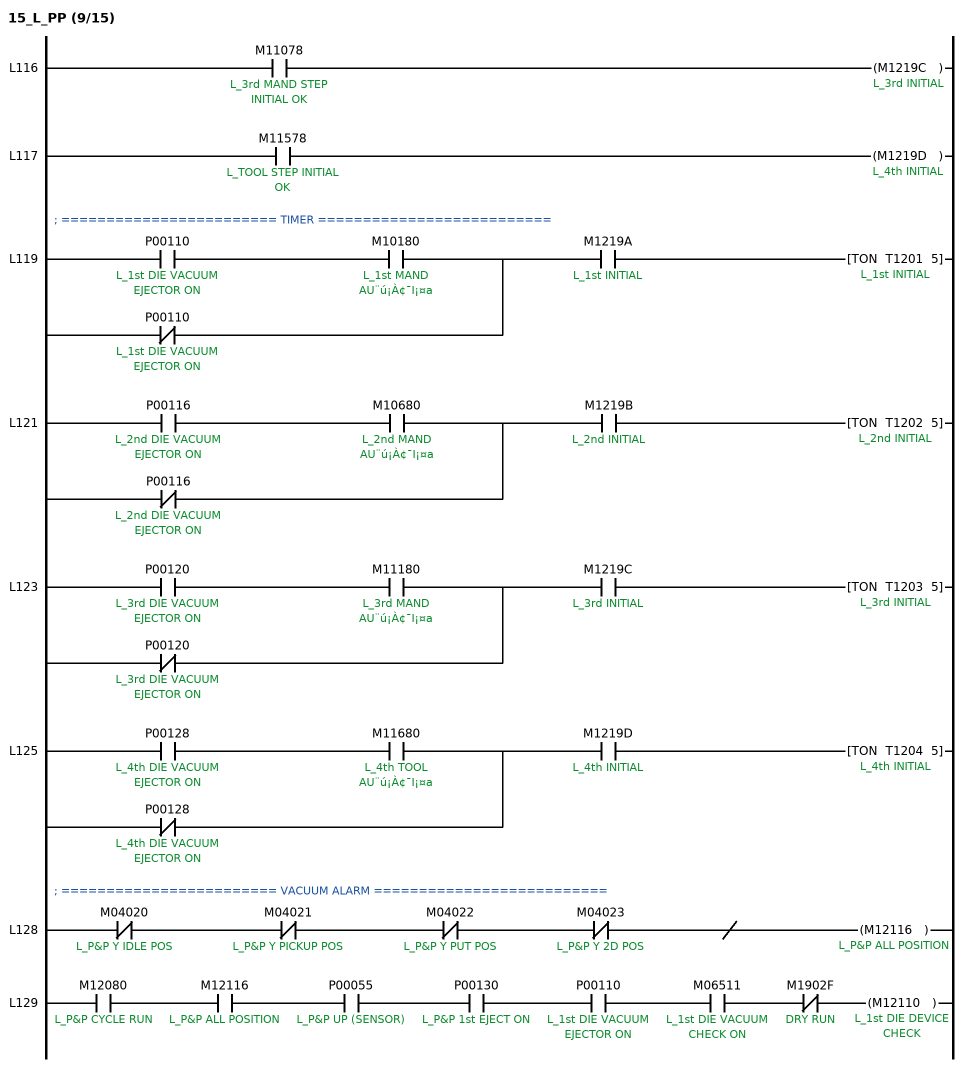
[picture p120: 15_L_PP rungs L116-L129]
; L116
LOAD      M11078	// L_3rd MAND STEP INITIAL OK
OUT       M1219C	// L_3rd INITIAL
; L117
LOAD      M11578	// L_TOOL STEP INITIAL OK
OUT       M1219D	// L_4th INITIAL
// ======================== TIMER ==========================
; L119
LOAD      P00110	// L_1st DIE VACUUM EJECTOR ON
AND       M10180	// L_1st MAND AU¨ú¡À¢¯I¡¤a
OR NOT    P00110	// L_1st DIE VACUUM EJECTOR ON
AND       M1219A	// L_1st INITIAL
TON       T1201 5	// L_1st INITIAL
; L121
LOAD      P00116	// L_2nd DIE VACUUM EJECTOR ON
AND       M10680	// L_2nd MAND AU¨ú¡À¢¯I¡¤a
OR NOT    P00116	// L_2nd DIE VACUUM EJECTOR ON
AND       M1219B	// L_2nd INITIAL
TON       T1202 5	// L_2nd INITIAL
; L123
LOAD      P00120	// L_3rd DIE VACUUM EJECTOR ON
AND       M11180	// L_3rd MAND AU¨ú¡À¢¯I¡¤a
OR NOT    P00120	// L_3rd DIE VACUUM EJECTOR ON
AND       M1219C	// L_3rd INITIAL
TON       T1203 5	// L_3rd INITIAL
; L125
LOAD      P00128	// L_4th DIE VACUUM EJECTOR ON
AND       M11680	// L_4th TOOL AU¨ú¡À¢¯I¡¤a
OR NOT    P00128	// L_4th DIE VACUUM EJECTOR ON
AND       M1219D	// L_4th INITIAL
TON       T1204 5	// L_4th INITIAL
// ======================== VACUUM ALARM ==========================
; L128
LOAD NOT  M04020	// L_P&P Y IDLE POS
AND NOT   M04021	// L_P&P Y PICKUP POS
AND NOT   M04022	// L_P&P Y PUT POS
AND NOT   M04023	// L_P&P Y 2D POS
NOT
OUT       M12116	// L_P&P ALL POSITION
; L129
LOAD      M12080	// L_P&P CYCLE RUN
AND       M12116	// L_P&P ALL POSITION
AND       P00055	// L_P&P UP (SENSOR)
AND       P00130	// L_P&P 1st EJECT ON
AND       P00110	// L_1st DIE VACUUM EJECTOR ON
AND       M06511	// L_1st DIE VACUUM CHECK ON
AND NOT   M1902F	// DRY RUN
OUT       M12110	// L_1st DIE DEVICE CHECK

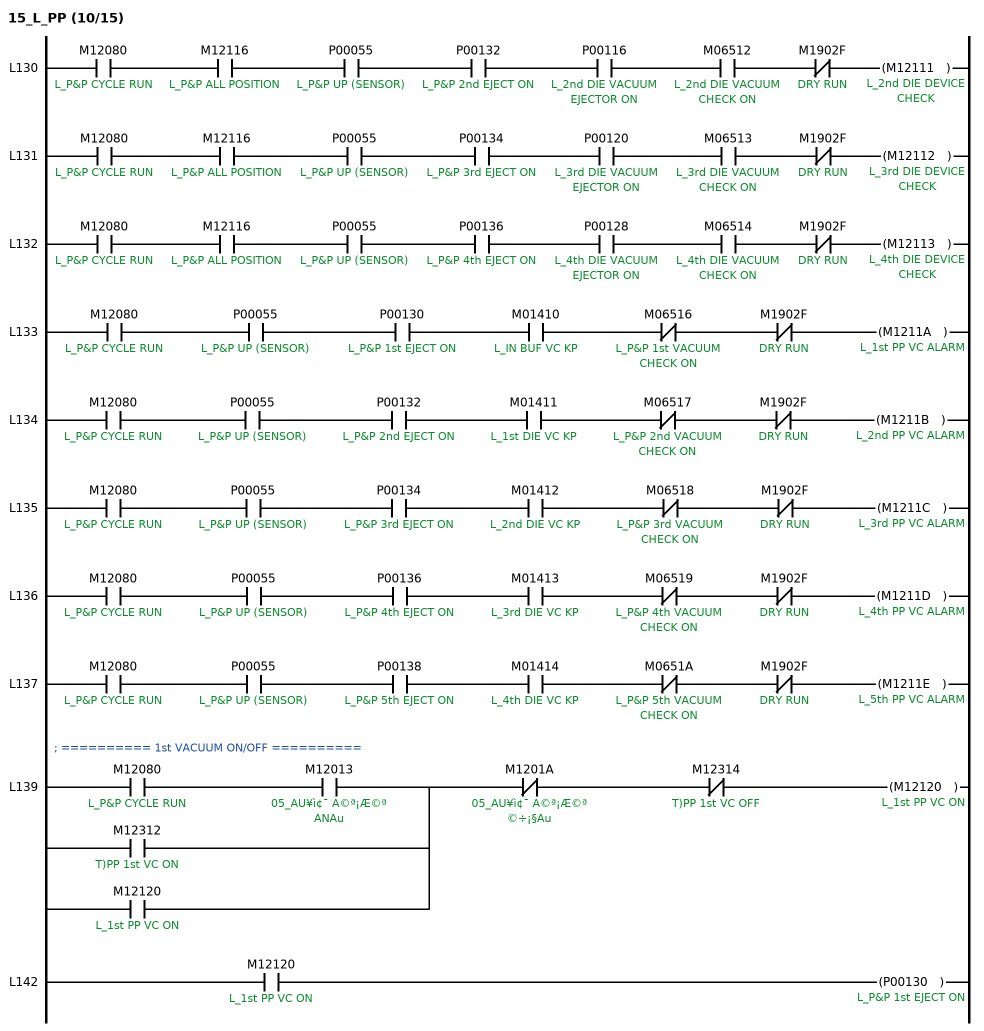
; L130
LOAD      M12080	// L_P&P CYCLE RUN
AND       M12116	// L_P&P ALL POSITION
AND       P00055	// L_P&P UP (SENSOR)
AND       P00132	// L_P&P 2nd EJECT ON
AND       P00116	// L_2nd DIE VACUUM EJECTOR ON
AND       M06512	// L_2nd DIE VACUUM CHECK ON
AND NOT   M1902F	// DRY RUN
OUT       M12111	// L_2nd DIE DEVICE CHECK
; L131
LOAD      M12080	// L_P&P CYCLE RUN
AND       M12116	// L_P&P ALL POSITION
AND       P00055	// L_P&P UP (SENSOR)
AND       P00134	// L_P&P 3rd EJECT ON
AND       P00120	// L_3rd DIE VACUUM EJECTOR ON
AND       M06513	// L_3rd DIE VACUUM CHECK ON
AND NOT   M1902F	// DRY RUN
OUT       M12112	// L_3rd DIE DEVICE CHECK
; L132
LOAD      M12080	// L_P&P CYCLE RUN
AND       M12116	// L_P&P ALL POSITION
AND       P00055	// L_P&P UP (SENSOR)
AND       P00136	// L_P&P 4th EJECT ON
AND       P00128	// L_4th DIE VACUUM EJECTOR ON
AND       M06514	// L_4th DIE VACUUM CHECK ON
AND NOT   M1902F	// DRY RUN
OUT       M12113	// L_4th DIE DEVICE CHECK
; L133
LOAD      M12080	// L_P&P CYCLE RUN
AND       P00055	// L_P&P UP (SENSOR)
AND       P00130	// L_P&P 1st EJECT ON
AND       M01410	// L_IN BUF VC KP
AND NOT   M06516	// L_P&P 1st VACUUM CHECK ON
AND NOT   M1902F	// DRY RUN
OUT       M1211A	// L_1st PP VC ALARM
; L134
LOAD      M12080	// L_P&P CYCLE RUN
AND       P00055	// L_P&P UP (SENSOR)
AND       P00132	// L_P&P 2nd EJECT ON
AND       M01411	// L_1st DIE VC KP
AND NOT   M06517	// L_P&P 2nd VACUUM CHECK ON
AND NOT   M1902F	// DRY RUN
OUT       M1211B	// L_2nd PP VC ALARM
; L135
LOAD      M12080	// L_P&P CYCLE RUN
AND       P00055	// L_P&P UP (SENSOR)
AND       P00134	// L_P&P 3rd EJECT ON
AND       M01412	// L_2nd DIE VC KP
AND NOT   M06518	// L_P&P 3rd VACUUM CHECK ON
AND NOT   M1902F	// DRY RUN
OUT       M1211C	// L_3rd PP VC ALARM
; L136
LOAD      M12080	// L_P&P CYCLE RUN
AND       P00055	// L_P&P UP (SENSOR)
AND       P00136	// L_P&P 4th EJECT ON
AND       M01413	// L_3rd DIE VC KP
AND NOT   M06519	// L_P&P 4th VACUUM CHECK ON
AND NOT   M1902F	// DRY RUN
OUT       M1211D	// L_4th PP VC ALARM
; L137
LOAD      M12080	// L_P&P CYCLE RUN
AND       P00055	// L_P&P UP (SENSOR)
AND       P00138	// L_P&P 5th EJECT ON
AND       M01414	// L_4th DIE VC KP
AND NOT   M0651A	// L_P&P 5th VACUUM CHECK ON
AND NOT   M1902F	// DRY RUN
OUT       M1211E	// L_5th PP VC ALARM
// ========== 1st VACUUM ON/OFF ==========
; L139
LOAD      M12080	// L_P&P CYCLE RUN
AND       M12013	// 05_AU¥ì¢¯ A©ª¡Æ©ª ANAu
OR        M12312	// T)PP 1st VC ON
OR        M12120	// L_1st PP VC ON
AND NOT   M1201A	// 05_AU¥ì¢¯ A©ª¡Æ©ª ©÷¡§Au
AND NOT   M12314	// T)PP 1st VC OFF
OUT       M12120	// L_1st PP VC ON
; L142
LOAD      M12120	// L_1st PP VC ON
OUT       P00130	// L_P&P 1st EJECT ON

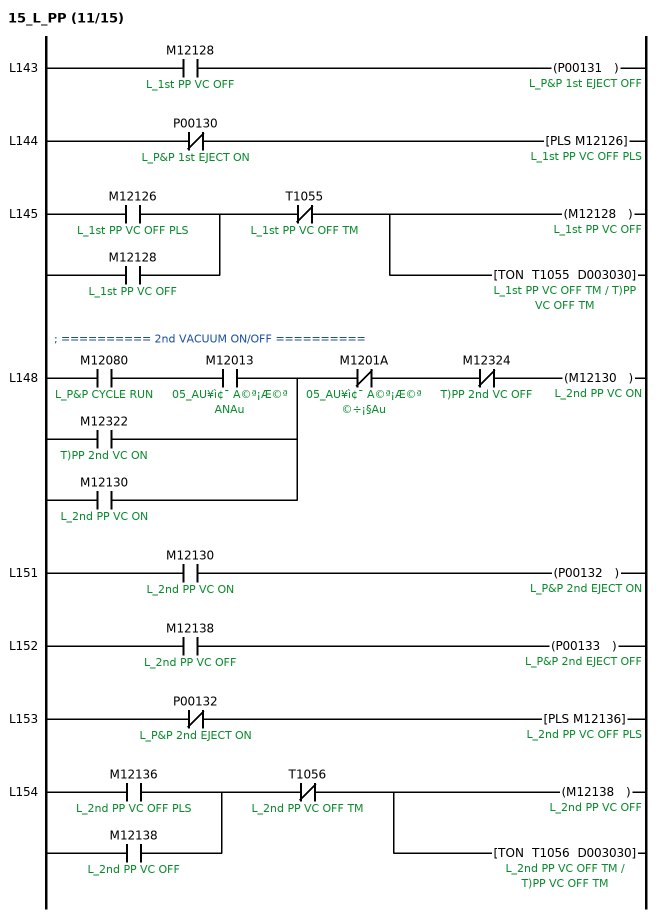
; L143
LOAD      M12128	// L_1st PP VC OFF
OUT       P00131	// L_P&P 1st EJECT OFF
; L144
LOAD NOT  P00130	// L_P&P 1st EJECT ON
OUTP      M12126	// L_1st PP VC OFF PLS
; L145
LOAD      M12126	// L_1st PP VC OFF PLS
OR        M12128	// L_1st PP VC OFF
AND NOT   T1055	// L_1st PP VC OFF TM
OUT       M12128	// L_1st PP VC OFF
TON       T1055 D003030	// L_1st PP VC OFF TM / T)PP VC OFF TM
// ========== 2nd VACUUM ON/OFF ==========
; L148
LOAD      M12080	// L_P&P CYCLE RUN
AND       M12013	// 05_AU¥ì¢¯ A©ª¡Æ©ª ANAu
OR        M12322	// T)PP 2nd VC ON
OR        M12130	// L_2nd PP VC ON
AND NOT   M1201A	// 05_AU¥ì¢¯ A©ª¡Æ©ª ©÷¡§Au
AND NOT   M12324	// T)PP 2nd VC OFF
OUT       M12130	// L_2nd PP VC ON
; L151
LOAD      M12130	// L_2nd PP VC ON
OUT       P00132	// L_P&P 2nd EJECT ON
; L152
LOAD      M12138	// L_2nd PP VC OFF
OUT       P00133	// L_P&P 2nd EJECT OFF
; L153
LOAD NOT  P00132	// L_P&P 2nd EJECT ON
OUTP      M12136	// L_2nd PP VC OFF PLS
; L154
LOAD      M12136	// L_2nd PP VC OFF PLS
OR        M12138	// L_2nd PP VC OFF
AND NOT   T1056	// L_2nd PP VC OFF TM
OUT       M12138	// L_2nd PP VC OFF
TON       T1056 D003030	// L_2nd PP VC OFF TM / T)PP VC OFF TM

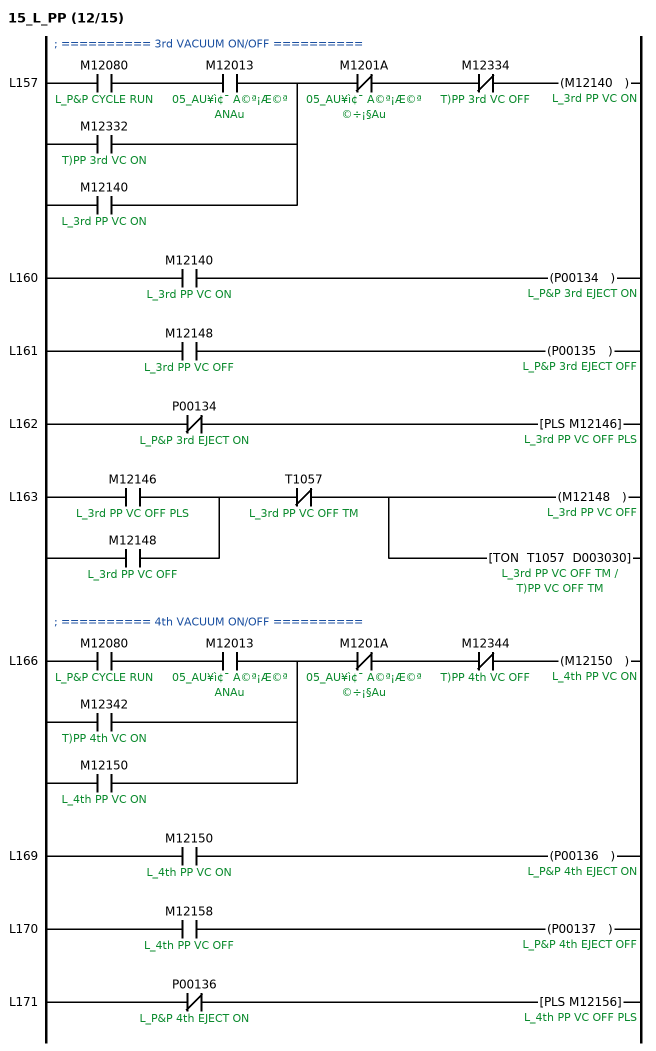
// ========== 3rd VACUUM ON/OFF ==========
; L157
LOAD      M12080	// L_P&P CYCLE RUN
AND       M12013	// 05_AU¥ì¢¯ A©ª¡Æ©ª ANAu
OR        M12332	// T)PP 3rd VC ON
OR        M12140	// L_3rd PP VC ON
AND NOT   M1201A	// 05_AU¥ì¢¯ A©ª¡Æ©ª ©÷¡§Au
AND NOT   M12334	// T)PP 3rd VC OFF
OUT       M12140	// L_3rd PP VC ON
; L160
LOAD      M12140	// L_3rd PP VC ON
OUT       P00134	// L_P&P 3rd EJECT ON
; L161
LOAD      M12148	// L_3rd PP VC OFF
OUT       P00135	// L_P&P 3rd EJECT OFF
; L162
LOAD NOT  P00134	// L_P&P 3rd EJECT ON
OUTP      M12146	// L_3rd PP VC OFF PLS
; L163
LOAD      M12146	// L_3rd PP VC OFF PLS
OR        M12148	// L_3rd PP VC OFF
AND NOT   T1057	// L_3rd PP VC OFF TM
OUT       M12148	// L_3rd PP VC OFF
TON       T1057 D003030	// L_3rd PP VC OFF TM / T)PP VC OFF TM
// ========== 4th VACUUM ON/OFF ==========
; L166
LOAD      M12080	// L_P&P CYCLE RUN
AND       M12013	// 05_AU¥ì¢¯ A©ª¡Æ©ª ANAu
OR        M12342	// T)PP 4th VC ON
OR        M12150	// L_4th PP VC ON
AND NOT   M1201A	// 05_AU¥ì¢¯ A©ª¡Æ©ª ©÷¡§Au
AND NOT   M12344	// T)PP 4th VC OFF
OUT       M12150	// L_4th PP VC ON
; L169
LOAD      M12150	// L_4th PP VC ON
OUT       P00136	// L_P&P 4th EJECT ON
; L170
LOAD      M12158	// L_4th PP VC OFF
OUT       P00137	// L_P&P 4th EJECT OFF
; L171
LOAD NOT  P00136	// L_P&P 4th EJECT ON
OUTP      M12156	// L_4th PP VC OFF PLS

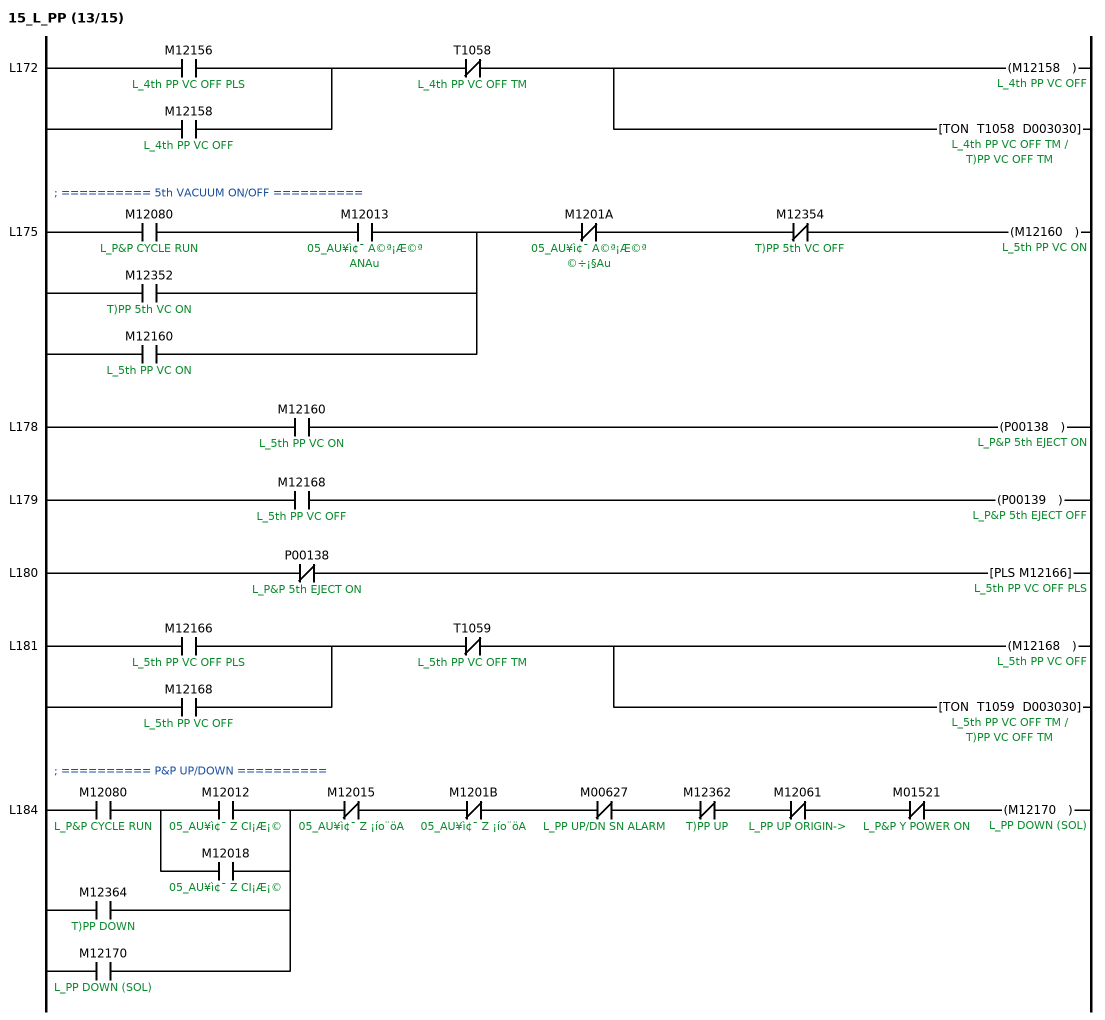
; L172
LOAD      M12156	// L_4th PP VC OFF PLS
OR        M12158	// L_4th PP VC OFF
AND NOT   T1058	// L_4th PP VC OFF TM
OUT       M12158	// L_4th PP VC OFF
TON       T1058 D003030	// L_4th PP VC OFF TM / T)PP VC OFF TM
// ========== 5th VACUUM ON/OFF ==========
; L175
LOAD      M12080	// L_P&P CYCLE RUN
AND       M12013	// 05_AU¥ì¢¯ A©ª¡Æ©ª ANAu
OR        M12352	// T)PP 5th VC ON
OR        M12160	// L_5th PP VC ON
AND NOT   M1201A	// 05_AU¥ì¢¯ A©ª¡Æ©ª ©÷¡§Au
AND NOT   M12354	// T)PP 5th VC OFF
OUT       M12160	// L_5th PP VC ON
; L178
LOAD      M12160	// L_5th PP VC ON
OUT       P00138	// L_P&P 5th EJECT ON
; L179
LOAD      M12168	// L_5th PP VC OFF
OUT       P00139	// L_P&P 5th EJECT OFF
; L180
LOAD NOT  P00138	// L_P&P 5th EJECT ON
OUTP      M12166	// L_5th PP VC OFF PLS
; L181
LOAD      M12166	// L_5th PP VC OFF PLS
OR        M12168	// L_5th PP VC OFF
AND NOT   T1059	// L_5th PP VC OFF TM
OUT       M12168	// L_5th PP VC OFF
TON       T1059 D003030	// L_5th PP VC OFF TM / T)PP VC OFF TM
// ========== P&P UP/DOWN ==========
; L184
LOAD      M12080	// L_P&P CYCLE RUN
LOAD      M12012	// 05_AU¥ì¢¯ Z CI¡Æ¡©
OR        M12018	// 05_AU¥ì¢¯ Z CI¡Æ¡©
AND LOAD
OR        M12364	// T)PP DOWN
OR        M12170	// L_PP DOWN (SOL)
AND NOT   M12015	// 05_AU¥ì¢¯ Z ¡ío¨öA
AND NOT   M1201B	// 05_AU¥ì¢¯ Z ¡ío¨öA
AND NOT   M00627	// L_PP UP/DN SN ALARM
AND NOT   M12362	// T)PP UP
AND NOT   M12061	// L_PP UP ORIGIN->
AND NOT   M01521	// L_P&P Y POWER ON
OUT       M12170	// L_PP DOWN (SOL)

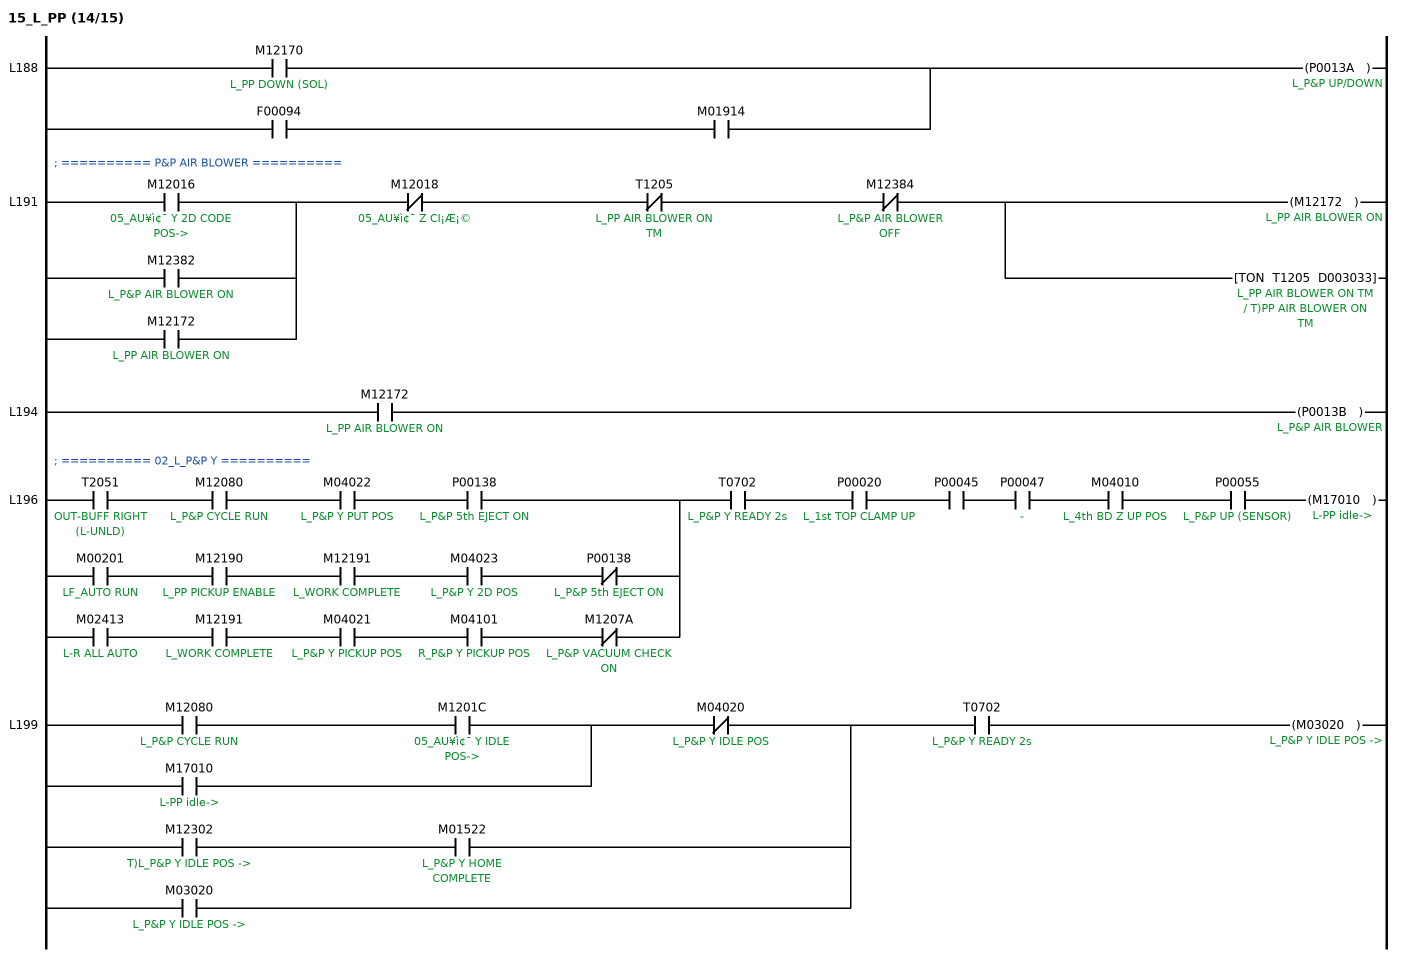
; L188
LOAD      M12170	// L_PP DOWN (SOL)
LOAD      F00094
AND       M01914
OR LOAD
OUT       P0013A	// L_P&P UP/DOWN
// ========== P&P AIR BLOWER ==========
; L191
LOAD      M12016	// 05_AU¥ì¢¯ Y 2D CODE POS->
OR        M12382	// L_P&P AIR BLOWER ON
OR        M12172	// L_PP AIR BLOWER ON
AND NOT   M12018	// 05_AU¥ì¢¯ Z CI¡Æ¡©
AND NOT   T1205	// L_PP AIR BLOWER ON TM
AND NOT   M12384	// L_P&P AIR BLOWER OFF
OUT       M12172	// L_PP AIR BLOWER ON
TON       T1205 D003033	// L_PP AIR BLOWER ON TM / T)PP AIR BLOWER ON TM
; L194
LOAD      M12172	// L_PP AIR BLOWER ON
OUT       P0013B	// L_P&P AIR BLOWER
// ========== 02_L_P&P Y ==========
; L196
LOAD      T2051	// OUT-BUFF RIGHT (L-UNLD)
AND       M12080	// L_P&P CYCLE RUN
AND       M04022	// L_P&P Y PUT POS
AND       P00138	// L_P&P 5th EJECT ON
LOAD      M00201	// LF_AUTO RUN
AND       M12190	// L_PP PICKUP ENABLE
AND       M12191	// L_WORK COMPLETE
AND       M04023	// L_P&P Y 2D POS
AND NOT   P00138	// L_P&P 5th EJECT ON
OR LOAD
LOAD      M02413	// L-R ALL AUTO
AND       M12191	// L_WORK COMPLETE
AND       M04021	// L_P&P Y PICKUP POS
AND       M04101	// R_P&P Y PICKUP POS
AND NOT   M1207A	// L_P&P VACUUM CHECK ON
OR LOAD
AND       T0702	// L_P&P Y READY 2s
AND       P00020	// L_1st TOP CLAMP UP
AND       P00045
AND       P00047	// -
AND       M04010	// L_4th BD Z UP POS
AND       P00055	// L_P&P UP (SENSOR)
OUT       M17010	// L-PP idle->
; L199
LOAD      M12080	// L_P&P CYCLE RUN
AND       M1201C	// 05_AU¥ì¢¯ Y IDLE POS->
OR        M17010	// L-PP idle->
AND NOT   M04020	// L_P&P Y IDLE POS
LOAD      M12302	// T)L_P&P Y IDLE POS ->
AND       M01522	// L_P&P Y HOME COMPLETE
OR LOAD
OR        M03020	// L_P&P Y IDLE POS ->
AND       T0702	// L_P&P Y READY 2s
OUT       M03020	// L_P&P Y IDLE POS ->

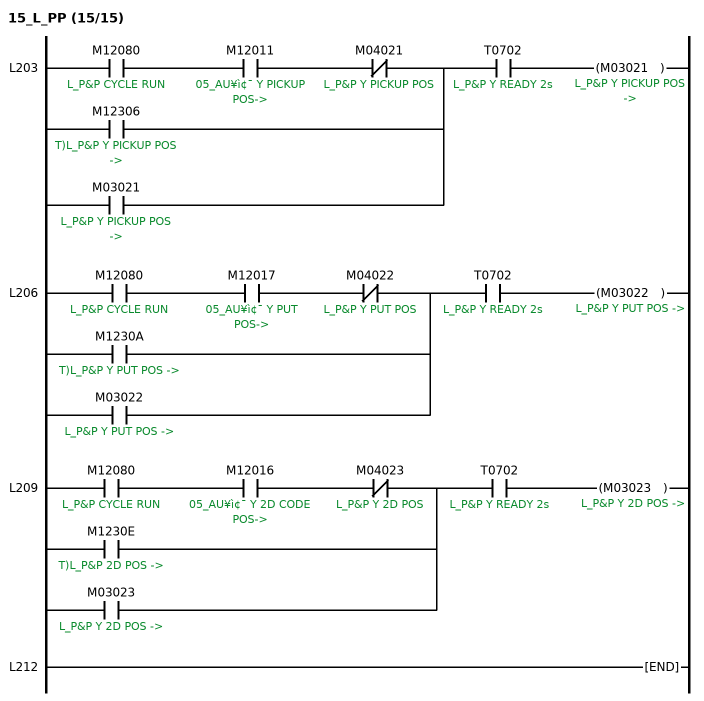
; L203
LOAD      M12080	// L_P&P CYCLE RUN
AND       M12011	// 05_AU¥ì¢¯ Y PICKUP POS->
AND NOT   M04021	// L_P&P Y PICKUP POS
OR        M12306	// T)L_P&P Y PICKUP POS ->
OR        M03021	// L_P&P Y PICKUP POS ->
AND       T0702	// L_P&P Y READY 2s
OUT       M03021	// L_P&P Y PICKUP POS ->
; L206
LOAD      M12080	// L_P&P CYCLE RUN
AND       M12017	// 05_AU¥ì¢¯ Y PUT POS->
AND NOT   M04022	// L_P&P Y PUT POS
OR        M1230A	// T)L_P&P Y PUT POS ->
OR        M03022	// L_P&P Y PUT POS ->
AND       T0702	// L_P&P Y READY 2s
OUT       M03022	// L_P&P Y PUT POS ->
; L209
LOAD      M12080	// L_P&P CYCLE RUN
AND       M12016	// 05_AU¥ì¢¯ Y 2D CODE POS->
AND NOT   M04023	// L_P&P Y 2D POS
OR        M1230E	// T)L_P&P 2D POS ->
OR        M03023	// L_P&P Y 2D POS ->
AND       T0702	// L_P&P Y READY 2s
OUT       M03023	// L_P&P Y 2D POS ->
; L212
END

PROGRAM 16_R_1st_MAND (task: ¨ö¨¬A¥ì CA¡¤I¡¾¡¿¡¤¡Í)

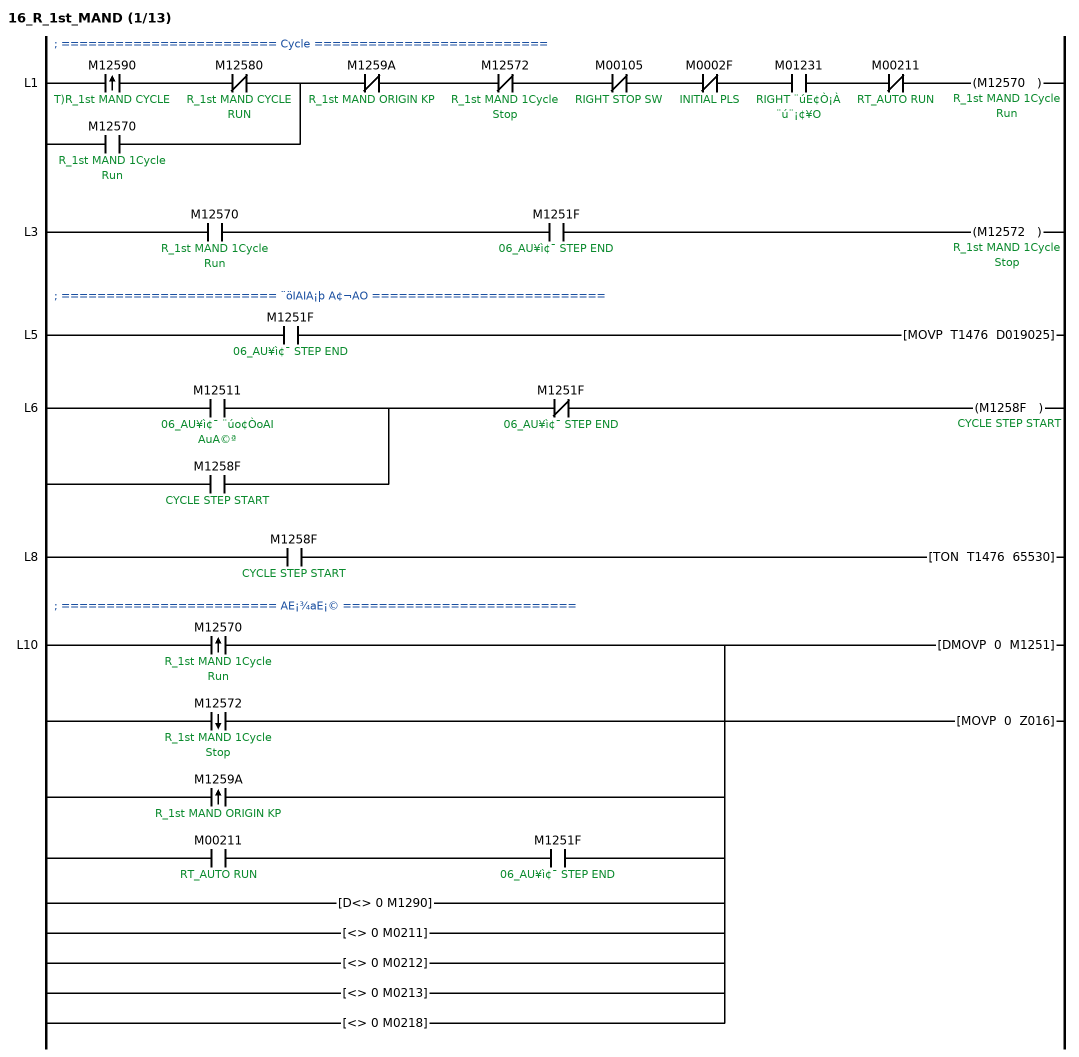
// ======================== Cycle ==========================
; L1
LOADP     M12590	// T)R_1st MAND CYCLE
AND NOT   M12580	// R_1st MAND CYCLE RUN
OR        M12570	// R_1st MAND 1Cycle Run
AND NOT   M1259A	// R_1st MAND ORIGIN KP
AND NOT   M12572	// R_1st MAND 1Cycle Stop
AND NOT   M00105	// RIGHT STOP SW
AND NOT   M0002F	// INITIAL PLS
AND       M01231	// RIGHT ¨úE¢Ò¡À ¨ú¨¡¢¥O
AND NOT   M00211	// RT_AUTO RUN
OUT       M12570	// R_1st MAND 1Cycle Run
; L3
LOAD      M12570	// R_1st MAND 1Cycle Run
AND       M1251F	// 06_AU¥ì¢¯ STEP END
OUT       M12572	// R_1st MAND 1Cycle Stop
// ======================== ¨öIAIA¡þ A¢¬AO ==========================
; L5
LOAD      M1251F	// 06_AU¥ì¢¯ STEP END
MOVP      T1476 D019025
; L6
LOAD      M12511	// 06_AU¥ì¢¯ ¨úo¢ÒoAI AuA©ª
OR        M1258F	// CYCLE STEP START
AND NOT   M1251F	// 06_AU¥ì¢¯ STEP END
OUT       M1258F	// CYCLE STEP START
; L8
LOAD      M1258F	// CYCLE STEP START
TON       T1476 65530
// ======================== AE¡¾aE¡© ==========================
; L10
LOADP     M12570	// R_1st MAND 1Cycle Run
ORN       M12572	// R_1st MAND 1Cycle Stop
ORP       M1259A	// R_1st MAND ORIGIN KP
LOAD      M00211	// RT_AUTO RUN
AND       M1251F	// 06_AU¥ì¢¯ STEP END
OR LOAD
ORD<>     0 M1290
OR<>      0 M0211
OR<>      0 M0212
OR<>      0 M0213
OR<>      0 M0218
DMOVP     0 M1251
MOVP      0 Z016

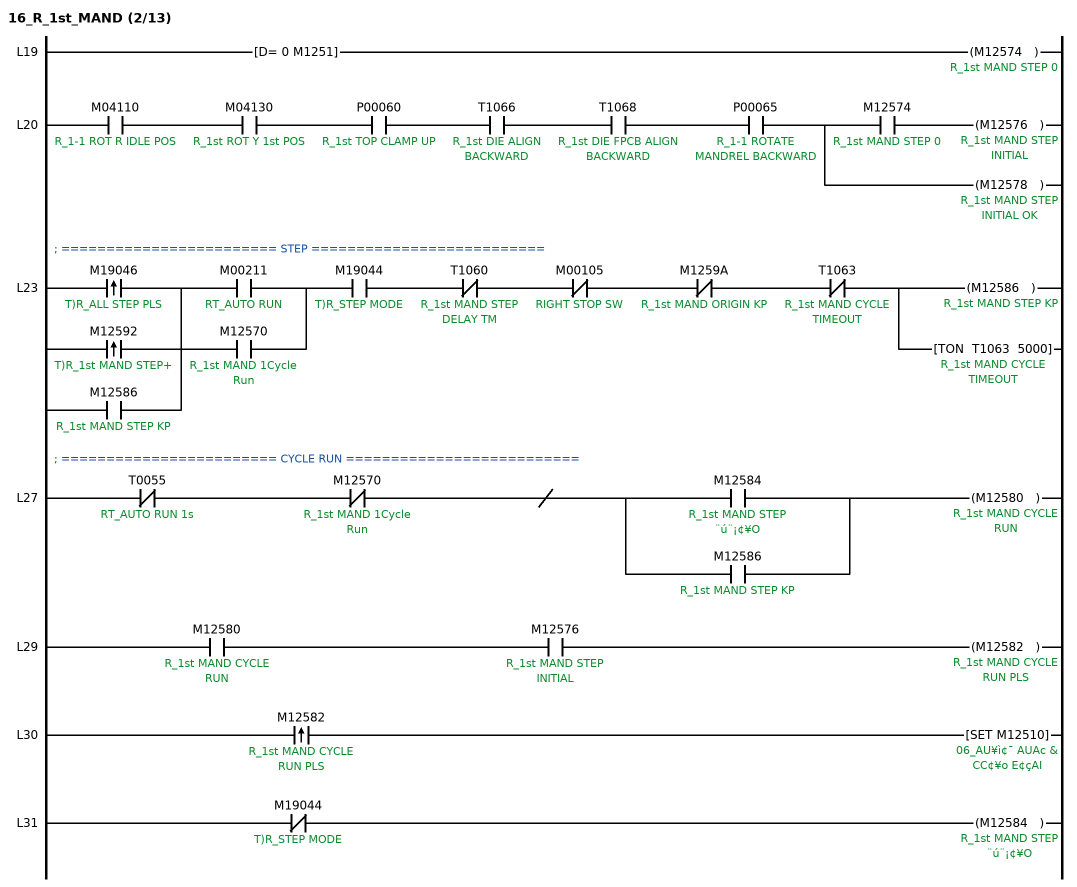
; L19
LOADD=    0 M1251
OUT       M12574	// R_1st MAND STEP 0
; L20
LOAD      M04110	// R_1-1 ROT R IDLE POS
AND       M04130	// R_1st ROT Y 1st POS
AND       P00060	// R_1st TOP CLAMP UP
AND       T1066	// R_1st DIE ALIGN BACKWARD
AND       T1068	// R_1st DIE FPCB ALIGN BACKWARD
AND       P00065	// R_1-1 ROTATE MANDREL BACKWARD
MPUSH
AND       M12574	// R_1st MAND STEP 0
OUT       M12576	// R_1st MAND STEP INITIAL
MPOP
OUT       M12578	// R_1st MAND STEP INITIAL OK
// ======================== STEP ==========================
; L23
LOADP     M19046	// T)R_ALL STEP PLS
ORP       M12592	// T)R_1st MAND STEP+
OR        M12586	// R_1st MAND STEP KP
LOAD      M00211	// RT_AUTO RUN
OR        M12570	// R_1st MAND 1Cycle Run
AND LOAD
AND       M19044	// T)R_STEP MODE
AND NOT   T1060	// R_1st MAND STEP DELAY TM
AND NOT   M00105	// RIGHT STOP SW
AND NOT   M1259A	// R_1st MAND ORIGIN KP
AND NOT   T1063	// R_1st MAND CYCLE TIMEOUT
OUT       M12586	// R_1st MAND STEP KP
TON       T1063 5000	// R_1st MAND CYCLE TIMEOUT
// ======================== CYCLE RUN ==========================
; L27
LOAD NOT  T0055	// RT_AUTO RUN 1s
AND NOT   M12570	// R_1st MAND 1Cycle Run
NOT
LOAD      M12584	// R_1st MAND STEP ¨ú¨¡¢¥O
OR        M12586	// R_1st MAND STEP KP
AND LOAD
OUT       M12580	// R_1st MAND CYCLE RUN
; L29
LOAD      M12580	// R_1st MAND CYCLE RUN
AND       M12576	// R_1st MAND STEP INITIAL
OUT       M12582	// R_1st MAND CYCLE RUN PLS
; L30
LOADP     M12582	// R_1st MAND CYCLE RUN PLS
SET       M12510	// 06_AU¥ì¢¯ AUAc & CC¢¥o E¢çAI
; L31
LOAD NOT  M19044	// T)R_STEP MODE
OUT       M12584	// R_1st MAND STEP ¨ú¨¡¢¥O

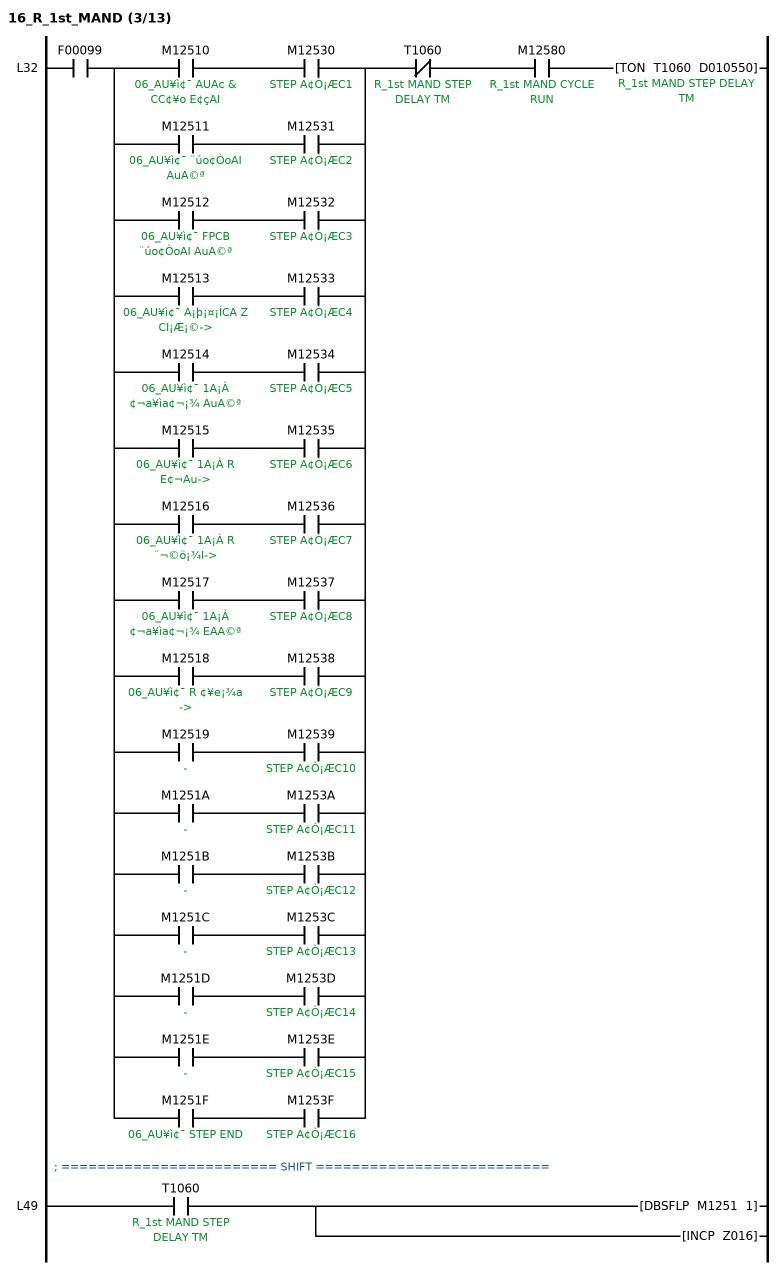
; L32
LOAD      F00099
LOAD      M12510	// 06_AU¥ì¢¯ AUAc & CC¢¥o E¢çAI
AND       M12530	// STEP A¢Ò¡ÆC1
LOAD      M12511	// 06_AU¥ì¢¯ ¨úo¢ÒoAI AuA©ª
AND       M12531	// STEP A¢Ò¡ÆC2
OR LOAD
LOAD      M12512	// 06_AU¥ì¢¯ FPCB ¨úo¢ÒoAI AuA©ª
AND       M12532	// STEP A¢Ò¡ÆC3
OR LOAD
LOAD      M12513	// 06_AU¥ì¢¯ A¡þ¡¤¡ÍCA Z CI¡Æ¡©->
AND       M12533	// STEP A¢Ò¡ÆC4
OR LOAD
LOAD      M12514	// 06_AU¥ì¢¯ 1A¡À ¢¬a¥ìa¢¬¡¾ AuA©ª
AND       M12534	// STEP A¢Ò¡ÆC5
OR LOAD
LOAD      M12515	// 06_AU¥ì¢¯ 1A¡À R E¢¬Au->
AND       M12535	// STEP A¢Ò¡ÆC6
OR LOAD
LOAD      M12516	// 06_AU¥ì¢¯ 1A¡À R ¨¬©ö¡¾I->
AND       M12536	// STEP A¢Ò¡ÆC7
OR LOAD
LOAD      M12517	// 06_AU¥ì¢¯ 1A¡À ¢¬a¥ìa¢¬¡¾ EAA©ª
AND       M12537	// STEP A¢Ò¡ÆC8
OR LOAD
LOAD      M12518	// 06_AU¥ì¢¯ R ¢¥e¡¾a ->
AND       M12538	// STEP A¢Ò¡ÆC9
OR LOAD
LOAD      M12519	// -
AND       M12539	// STEP A¢Ò¡ÆC10
OR LOAD
LOAD      M1251A	// -
AND       M1253A	// STEP A¢Ò¡ÆC11
OR LOAD
LOAD      M1251B	// -
AND       M1253B	// STEP A¢Ò¡ÆC12
OR LOAD
LOAD      M1251C	// -
AND       M1253C	// STEP A¢Ò¡ÆC13
OR LOAD
LOAD      M1251D	// -
AND       M1253D	// STEP A¢Ò¡ÆC14
OR LOAD
LOAD      M1251E	// -
AND       M1253E	// STEP A¢Ò¡ÆC15
OR LOAD
LOAD      M1251F	// 06_AU¥ì¢¯ STEP END
AND       M1253F	// STEP A¢Ò¡ÆC16
OR LOAD
AND LOAD
AND NOT   T1060	// R_1st MAND STEP DELAY TM
AND       M12580	// R_1st MAND CYCLE RUN
TON       T1060 D010550	// R_1st MAND STEP DELAY TM
// ======================== SHIFT ==========================
; L49
LOAD      T1060	// R_1st MAND STEP DELAY TM
DBSFLP    M1251 1
INCP      Z016

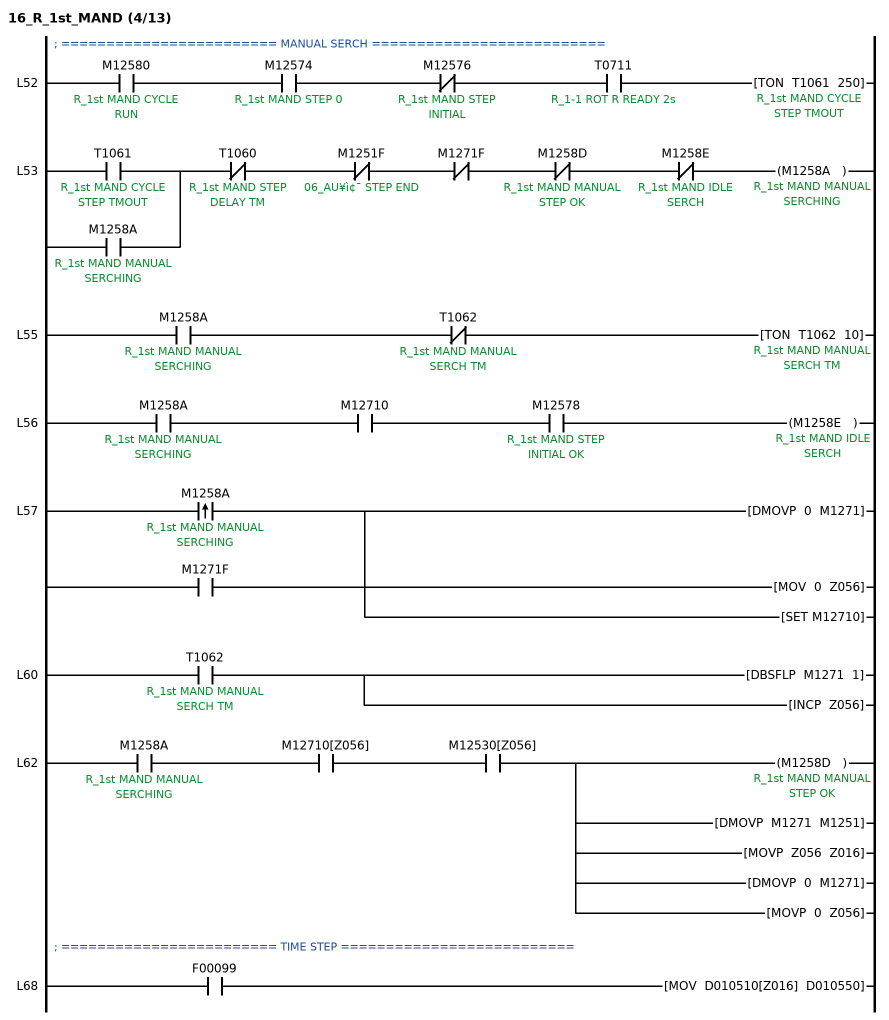
// ======================== MANUAL SERCH ==========================
; L52
LOAD      M12580	// R_1st MAND CYCLE RUN
AND       M12574	// R_1st MAND STEP 0
AND NOT   M12576	// R_1st MAND STEP INITIAL
AND       T0711	// R_1-1 ROT R READY 2s
TON       T1061 250	// R_1st MAND CYCLE STEP TMOUT
; L53
LOAD      T1061	// R_1st MAND CYCLE STEP TMOUT
OR        M1258A	// R_1st MAND MANUAL SERCHING
AND NOT   T1060	// R_1st MAND STEP DELAY TM
AND NOT   M1251F	// 06_AU¥ì¢¯ STEP END
AND NOT   M1271F
AND NOT   M1258D	// R_1st MAND MANUAL STEP OK
AND NOT   M1258E	// R_1st MAND IDLE SERCH
OUT       M1258A	// R_1st MAND MANUAL SERCHING
; L55
LOAD      M1258A	// R_1st MAND MANUAL SERCHING
AND NOT   T1062	// R_1st MAND MANUAL SERCH TM
TON       T1062 10	// R_1st MAND MANUAL SERCH TM
; L56
LOAD      M1258A	// R_1st MAND MANUAL SERCHING
AND       M12710
AND       M12578	// R_1st MAND STEP INITIAL OK
OUT       M1258E	// R_1st MAND IDLE SERCH
; L57
LOADP     M1258A	// R_1st MAND MANUAL SERCHING
OR        M1271F
DMOVP     0 M1271
MOV       0 Z056
SET       M12710
; L60
LOAD      T1062	// R_1st MAND MANUAL SERCH TM
DBSFLP    M1271 1
INCP      Z056
; L62
LOAD      M1258A	// R_1st MAND MANUAL SERCHING
AND       M12710[Z056]
AND       M12530[Z056]
OUT       M1258D	// R_1st MAND MANUAL STEP OK
DMOVP     M1271 M1251
MOVP      Z056 Z016
DMOVP     0 M1271
MOVP      0 Z056
// ======================== TIME STEP ==========================
; L68
LOAD      F00099
MOV       D010510[Z016] D010550

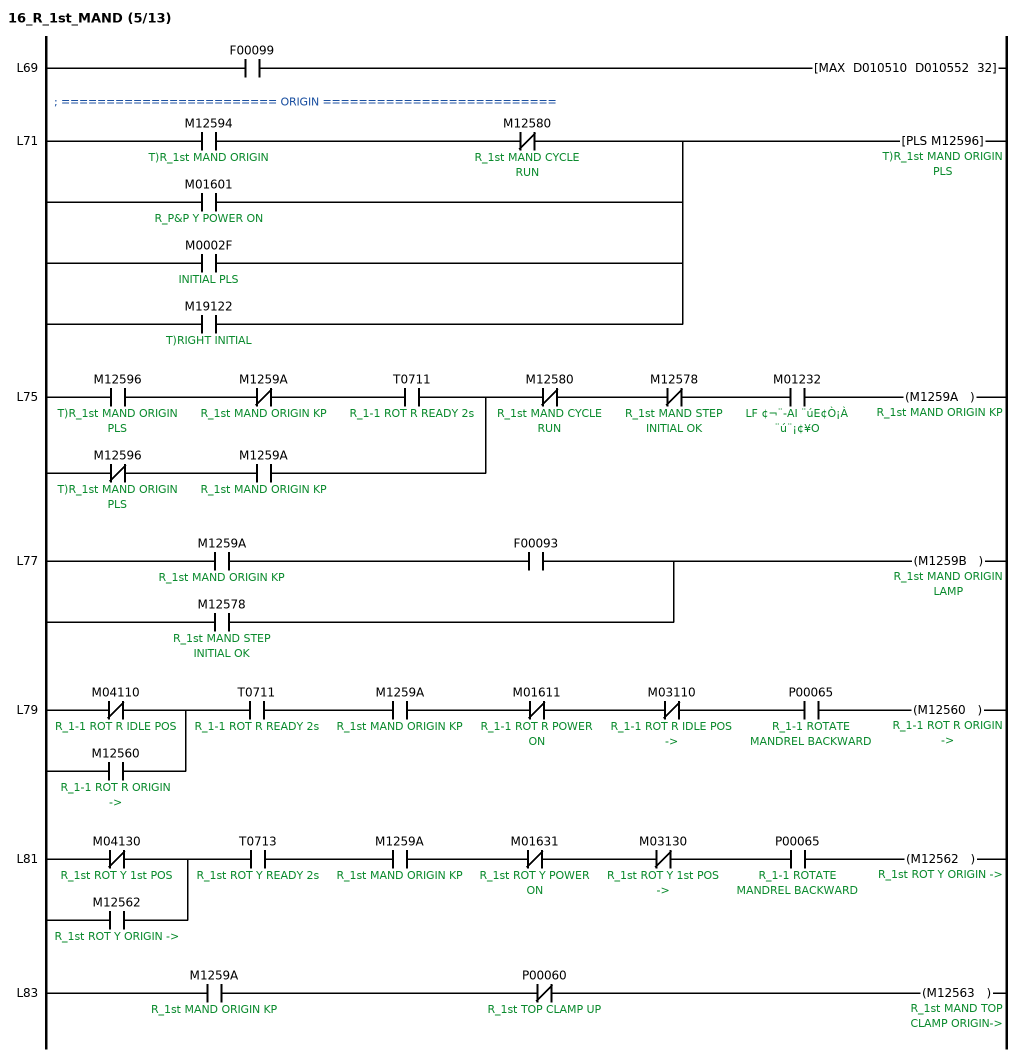
; L69
LOAD      F00099
MAX       D010510 D010552 32
// ======================== ORIGIN ==========================
; L71
LOAD      M12594	// T)R_1st MAND ORIGIN
AND NOT   M12580	// R_1st MAND CYCLE RUN
OR        M01601	// R_P&P Y POWER ON
OR        M0002F	// INITIAL PLS
OR        M19122	// T)RIGHT INITIAL
OUTP      M12596	// T)R_1st MAND ORIGIN PLS
; L75
LOAD      M12596	// T)R_1st MAND ORIGIN PLS
AND NOT   M1259A	// R_1st MAND ORIGIN KP
AND       T0711	// R_1-1 ROT R READY 2s
LOAD NOT  M12596	// T)R_1st MAND ORIGIN PLS
AND       M1259A	// R_1st MAND ORIGIN KP
OR LOAD
AND NOT   M12580	// R_1st MAND CYCLE RUN
AND NOT   M12578	// R_1st MAND STEP INITIAL OK
AND       M01232	// LF ¢¬¨­AI ¨úE¢Ò¡À ¨ú¨¡¢¥O
OUT       M1259A	// R_1st MAND ORIGIN KP
; L77
LOAD      M1259A	// R_1st MAND ORIGIN KP
AND       F00093
OR        M12578	// R_1st MAND STEP INITIAL OK
OUT       M1259B	// R_1st MAND ORIGIN LAMP
; L79
LOAD NOT  M04110	// R_1-1 ROT R IDLE POS
OR        M12560	// R_1-1 ROT R ORIGIN ->
AND       T0711	// R_1-1 ROT R READY 2s
AND       M1259A	// R_1st MAND ORIGIN KP
AND NOT   M01611	// R_1-1 ROT R POWER ON
AND NOT   M03110	// R_1-1 ROT R IDLE POS ->
AND       P00065	// R_1-1 ROTATE MANDREL BACKWARD
OUT       M12560	// R_1-1 ROT R ORIGIN ->
; L81
LOAD NOT  M04130	// R_1st ROT Y 1st POS
OR        M12562	// R_1st ROT Y ORIGIN ->
AND       T0713	// R_1st ROT Y READY 2s
AND       M1259A	// R_1st MAND ORIGIN KP
AND NOT   M01631	// R_1st ROT Y POWER ON
AND NOT   M03130	// R_1st ROT Y 1st POS ->
AND       P00065	// R_1-1 ROTATE MANDREL BACKWARD
OUT       M12562	// R_1st ROT Y ORIGIN ->
; L83
LOAD      M1259A	// R_1st MAND ORIGIN KP
AND NOT   P00060	// R_1st TOP CLAMP UP
OUT       M12563	// R_1st MAND TOP CLAMP ORIGIN->

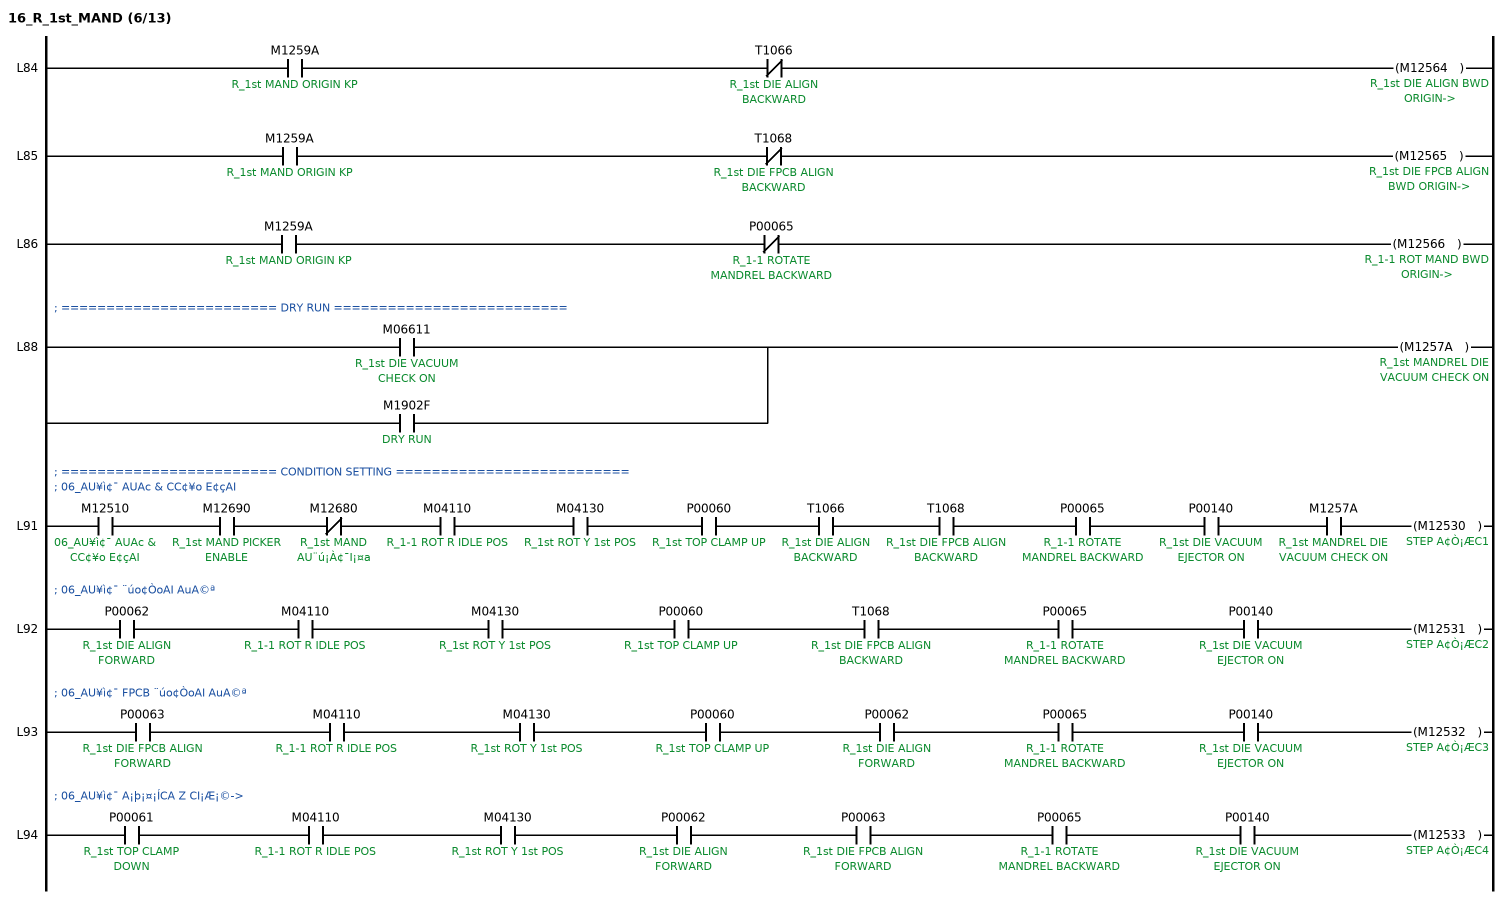
; L84
LOAD      M1259A	// R_1st MAND ORIGIN KP
AND NOT   T1066	// R_1st DIE ALIGN BACKWARD
OUT       M12564	// R_1st DIE ALIGN BWD ORIGIN->
; L85
LOAD      M1259A	// R_1st MAND ORIGIN KP
AND NOT   T1068	// R_1st DIE FPCB ALIGN BACKWARD
OUT       M12565	// R_1st DIE FPCB ALIGN BWD ORIGIN->
; L86
LOAD      M1259A	// R_1st MAND ORIGIN KP
AND NOT   P00065	// R_1-1 ROTATE MANDREL BACKWARD
OUT       M12566	// R_1-1 ROT MAND BWD ORIGIN->
// ======================== DRY RUN ==========================
; L88
LOAD      M06611	// R_1st DIE VACUUM CHECK ON
OR        M1902F	// DRY RUN
OUT       M1257A	// R_1st MANDREL DIE VACUUM CHECK ON
// ======================== CONDITION SETTING ==========================
; L91
LOAD      M12510	// 06_AU¥ì¢¯ AUAc & CC¢¥o E¢çAI
AND       M12690	// R_1st MAND PICKER ENABLE
AND NOT   M12680	// R_1st MAND AU¨ú¡À¢¯I¡¤a
AND       M04110	// R_1-1 ROT R IDLE POS
AND       M04130	// R_1st ROT Y 1st POS
AND       P00060	// R_1st TOP CLAMP UP
AND       T1066	// R_1st DIE ALIGN BACKWARD
AND       T1068	// R_1st DIE FPCB ALIGN BACKWARD
AND       P00065	// R_1-1 ROTATE MANDREL BACKWARD
AND       P00140	// R_1st DIE VACUUM EJECTOR ON
AND       M1257A	// R_1st MANDREL DIE VACUUM CHECK ON
OUT       M12530	// STEP A¢Ò¡ÆC1
// output comment: 06_AU¥ì¢¯ AUAc & CC¢¥o E¢çAI
; L92
LOAD      P00062	// R_1st DIE ALIGN FORWARD
AND       M04110	// R_1-1 ROT R IDLE POS
AND       M04130	// R_1st ROT Y 1st POS
AND       P00060	// R_1st TOP CLAMP UP
AND       T1068	// R_1st DIE FPCB ALIGN BACKWARD
AND       P00065	// R_1-1 ROTATE MANDREL BACKWARD
AND       P00140	// R_1st DIE VACUUM EJECTOR ON
OUT       M12531	// STEP A¢Ò¡ÆC2
// output comment: 06_AU¥ì¢¯ ¨úo¢ÒoAI AuA©ª
; L93
LOAD      P00063	// R_1st DIE FPCB ALIGN FORWARD
AND       M04110	// R_1-1 ROT R IDLE POS
AND       M04130	// R_1st ROT Y 1st POS
AND       P00060	// R_1st TOP CLAMP UP
AND       P00062	// R_1st DIE ALIGN FORWARD
AND       P00065	// R_1-1 ROTATE MANDREL BACKWARD
AND       P00140	// R_1st DIE VACUUM EJECTOR ON
OUT       M12532	// STEP A¢Ò¡ÆC3
// output comment: 06_AU¥ì¢¯ FPCB ¨úo¢ÒoAI AuA©ª
; L94
LOAD      P00061	// R_1st TOP CLAMP DOWN
AND       M04110	// R_1-1 ROT R IDLE POS
AND       M04130	// R_1st ROT Y 1st POS
AND       P00062	// R_1st DIE ALIGN FORWARD
AND       P00063	// R_1st DIE FPCB ALIGN FORWARD
AND       P00065	// R_1-1 ROTATE MANDREL BACKWARD
AND       P00140	// R_1st DIE VACUUM EJECTOR ON
OUT       M12533	// STEP A¢Ò¡ÆC4
// output comment: 06_AU¥ì¢¯ A¡þ¡¤¡ÍCA Z CI¡Æ¡©->

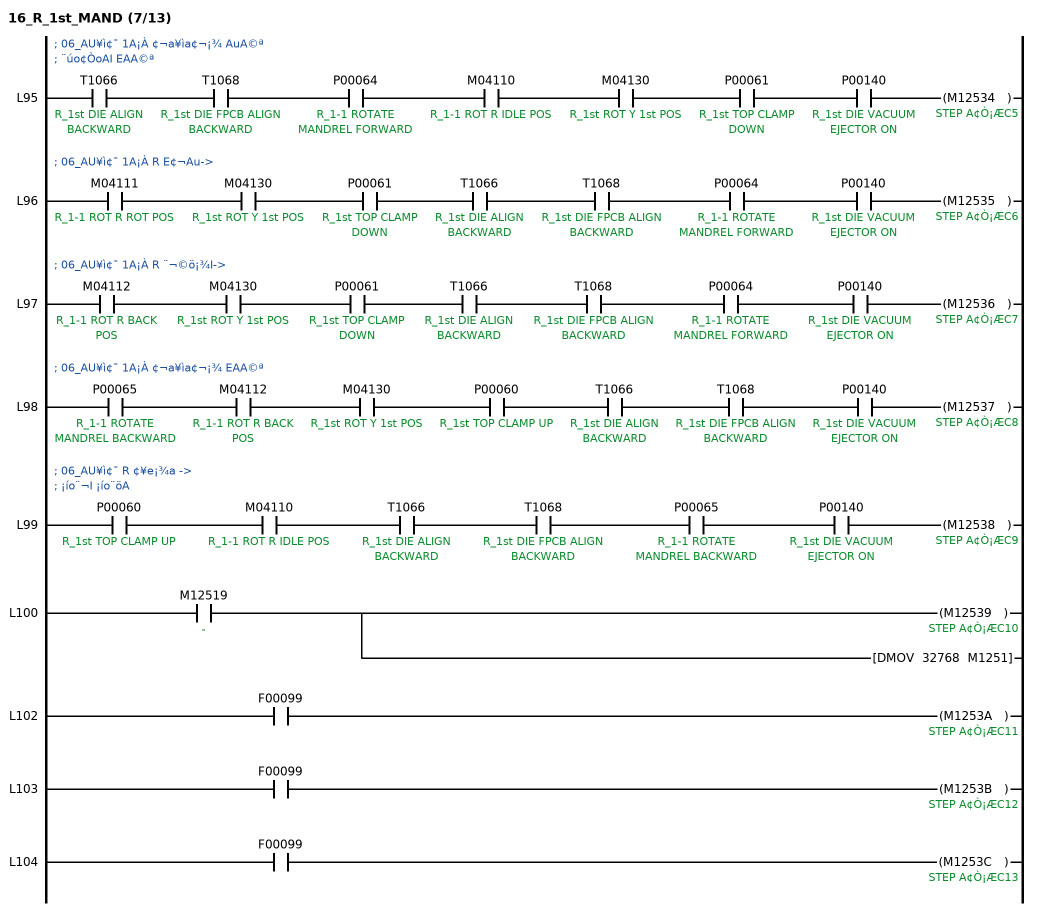
; L95
LOAD      T1066	// R_1st DIE ALIGN BACKWARD
AND       T1068	// R_1st DIE FPCB ALIGN BACKWARD
AND       P00064	// R_1-1 ROTATE MANDREL FORWARD
AND       M04110	// R_1-1 ROT R IDLE POS
AND       M04130	// R_1st ROT Y 1st POS
AND       P00061	// R_1st TOP CLAMP DOWN
AND       P00140	// R_1st DIE VACUUM EJECTOR ON
OUT       M12534	// STEP A¢Ò¡ÆC5
// output comment: 06_AU¥ì¢¯ 1A¡À ¢¬a¥ìa¢¬¡¾ AuA©ª ¨úo¢ÒoAI EAA©ª
; L96
LOAD      M04111	// R_1-1 ROT R ROT POS
AND       M04130	// R_1st ROT Y 1st POS
AND       P00061	// R_1st TOP CLAMP DOWN
AND       T1066	// R_1st DIE ALIGN BACKWARD
AND       T1068	// R_1st DIE FPCB ALIGN BACKWARD
AND       P00064	// R_1-1 ROTATE MANDREL FORWARD
AND       P00140	// R_1st DIE VACUUM EJECTOR ON
OUT       M12535	// STEP A¢Ò¡ÆC6
// output comment: 06_AU¥ì¢¯ 1A¡À R E¢¬Au->
; L97
LOAD      M04112	// R_1-1 ROT R BACK POS
AND       M04130	// R_1st ROT Y 1st POS
AND       P00061	// R_1st TOP CLAMP DOWN
AND       T1066	// R_1st DIE ALIGN BACKWARD
AND       T1068	// R_1st DIE FPCB ALIGN BACKWARD
AND       P00064	// R_1-1 ROTATE MANDREL FORWARD
AND       P00140	// R_1st DIE VACUUM EJECTOR ON
OUT       M12536	// STEP A¢Ò¡ÆC7
// output comment: 06_AU¥ì¢¯ 1A¡À R ¨¬©ö¡¾I->
; L98
LOAD      P00065	// R_1-1 ROTATE MANDREL BACKWARD
AND       M04112	// R_1-1 ROT R BACK POS
AND       M04130	// R_1st ROT Y 1st POS
AND       P00060	// R_1st TOP CLAMP UP
AND       T1066	// R_1st DIE ALIGN BACKWARD
AND       T1068	// R_1st DIE FPCB ALIGN BACKWARD
AND       P00140	// R_1st DIE VACUUM EJECTOR ON
OUT       M12537	// STEP A¢Ò¡ÆC8
// output comment: 06_AU¥ì¢¯ 1A¡À ¢¬a¥ìa¢¬¡¾ EAA©ª
; L99
LOAD      P00060	// R_1st TOP CLAMP UP
AND       M04110	// R_1-1 ROT R IDLE POS
AND       T1066	// R_1st DIE ALIGN BACKWARD
AND       T1068	// R_1st DIE FPCB ALIGN BACKWARD
AND       P00065	// R_1-1 ROTATE MANDREL BACKWARD
AND       P00140	// R_1st DIE VACUUM EJECTOR ON
OUT       M12538	// STEP A¢Ò¡ÆC9
// output comment: 06_AU¥ì¢¯ R ¢¥e¡¾a -> ¡ío¨¬I ¡ío¨öA
; L100
LOAD      M12519	// -
OUT       M12539	// STEP A¢Ò¡ÆC10
DMOV      32768 M1251
; L102
LOAD      F00099
OUT       M1253A	// STEP A¢Ò¡ÆC11
; L103
LOAD      F00099
OUT       M1253B	// STEP A¢Ò¡ÆC12
; L104
LOAD      F00099
OUT       M1253C	// STEP A¢Ò¡ÆC13

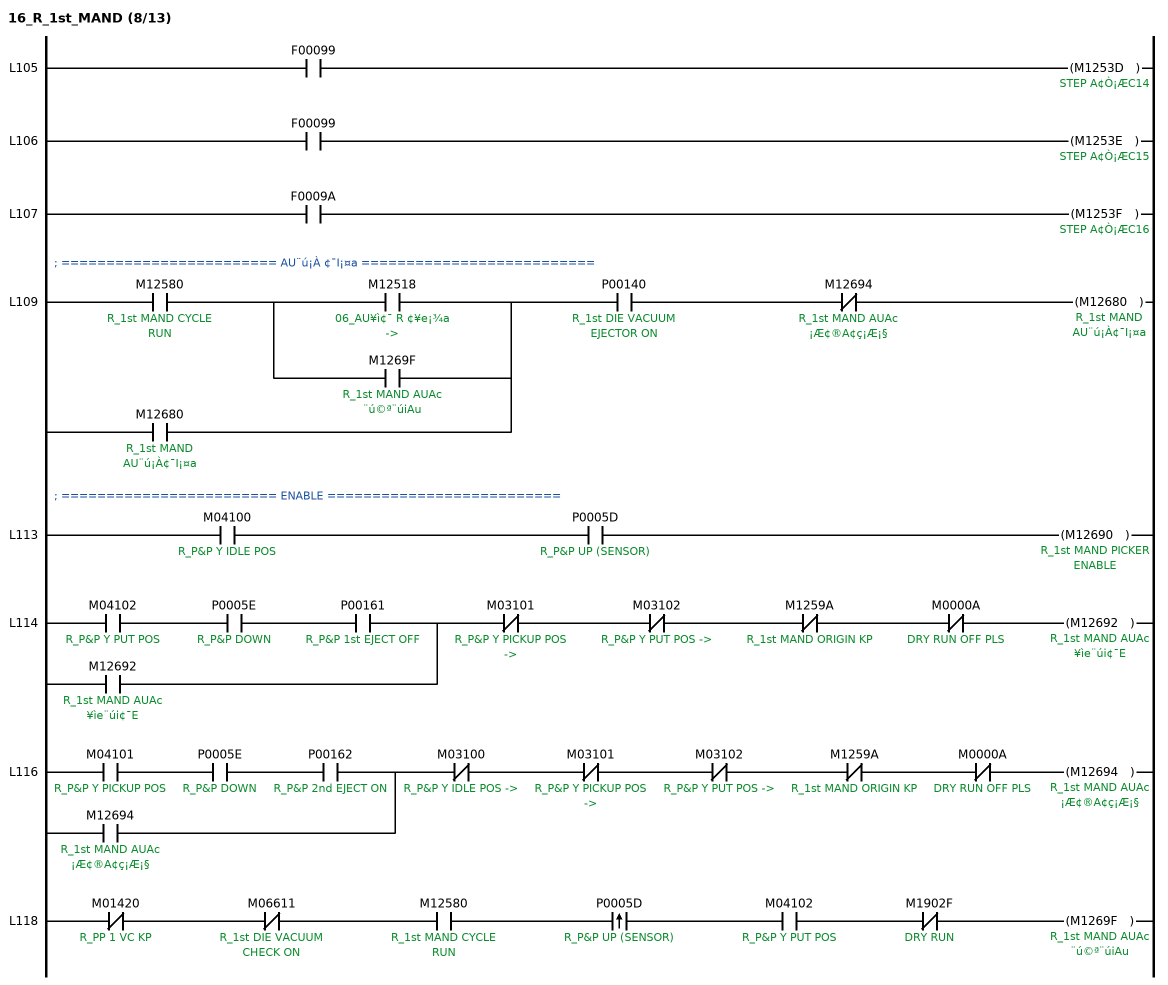
; L105
LOAD      F00099
OUT       M1253D	// STEP A¢Ò¡ÆC14
; L106
LOAD      F00099
OUT       M1253E	// STEP A¢Ò¡ÆC15
; L107
LOAD      F0009A
OUT       M1253F	// STEP A¢Ò¡ÆC16
// ======================== AU¨ú¡À ¢¯I¡¤a ==========================
; L109
LOAD      M12580	// R_1st MAND CYCLE RUN
LOAD      M12518	// 06_AU¥ì¢¯ R ¢¥e¡¾a ->
OR        M1269F	// R_1st MAND AUAc ¨ú©ª¨úiAu
AND LOAD
OR        M12680	// R_1st MAND AU¨ú¡À¢¯I¡¤a
AND       P00140	// R_1st DIE VACUUM EJECTOR ON
AND NOT   M12694	// R_1st MAND AUAc ¡Æ¢®A¢ç¡Æ¡§
OUT       M12680	// R_1st MAND AU¨ú¡À¢¯I¡¤a
// ======================== ENABLE ==========================
; L113
LOAD      M04100	// R_P&P Y IDLE POS
AND       P0005D	// R_P&P UP (SENSOR)
OUT       M12690	// R_1st MAND PICKER ENABLE
; L114
LOAD      M04102	// R_P&P Y PUT POS
AND       P0005E	// R_P&P DOWN
AND       P00161	// R_P&P 1st EJECT OFF
OR        M12692	// R_1st MAND AUAc ¥ìe¨úi¢¯E
AND NOT   M03101	// R_P&P Y PICKUP POS ->
AND NOT   M03102	// R_P&P Y PUT POS ->
AND NOT   M1259A	// R_1st MAND ORIGIN KP
AND NOT   M0000A	// DRY RUN OFF PLS
OUT       M12692	// R_1st MAND AUAc ¥ìe¨úi¢¯E
; L116
LOAD      M04101	// R_P&P Y PICKUP POS
AND       P0005E	// R_P&P DOWN
AND       P00162	// R_P&P 2nd EJECT ON
OR        M12694	// R_1st MAND AUAc ¡Æ¢®A¢ç¡Æ¡§
AND NOT   M03100	// R_P&P Y IDLE POS ->
AND NOT   M03101	// R_P&P Y PICKUP POS ->
AND NOT   M03102	// R_P&P Y PUT POS ->
AND NOT   M1259A	// R_1st MAND ORIGIN KP
AND NOT   M0000A	// DRY RUN OFF PLS
OUT       M12694	// R_1st MAND AUAc ¡Æ¢®A¢ç¡Æ¡§
; L118
LOAD NOT  M01420	// R_PP 1 VC KP
AND NOT   M06611	// R_1st DIE VACUUM CHECK ON
AND       M12580	// R_1st MAND CYCLE RUN
ANDP      P0005D	// R_P&P UP (SENSOR)
AND       M04102	// R_P&P Y PUT POS
AND NOT   M1902F	// DRY RUN
OUT       M1269F	// R_1st MAND AUAc ¨ú©ª¨úiAu

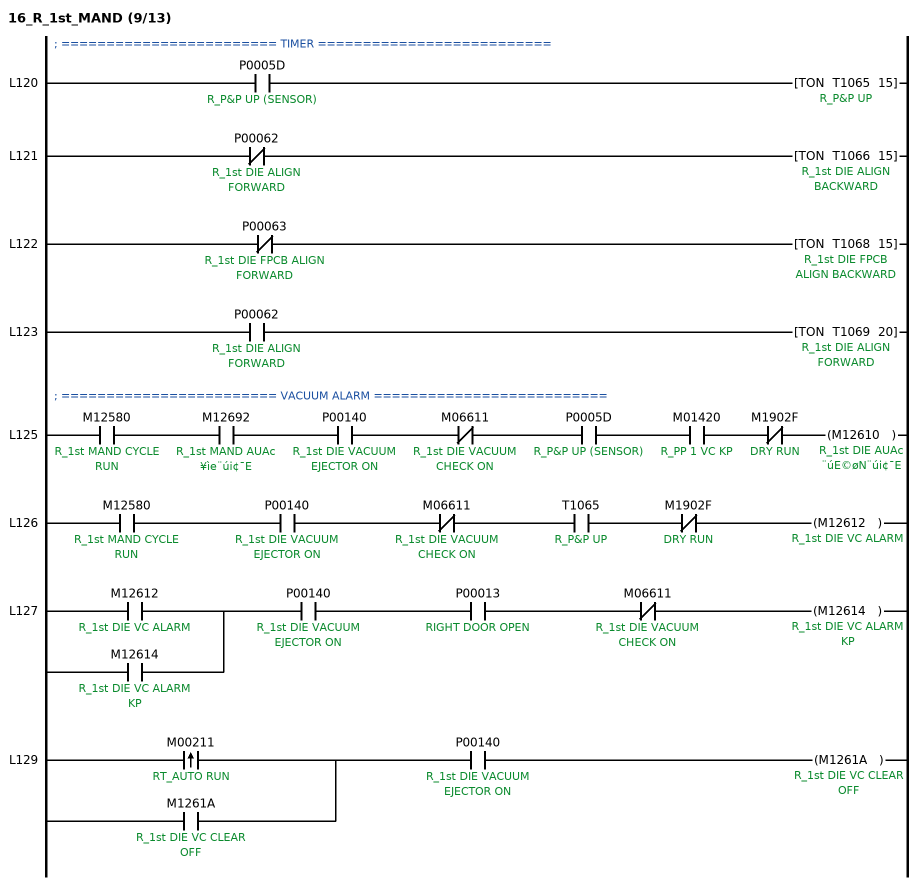
// ======================== TIMER ==========================
; L120
LOAD      P0005D	// R_P&P UP (SENSOR)
TON       T1065 15	// R_P&P UP
; L121
LOAD NOT  P00062	// R_1st DIE ALIGN FORWARD
TON       T1066 15	// R_1st DIE ALIGN BACKWARD
; L122
LOAD NOT  P00063	// R_1st DIE FPCB ALIGN FORWARD
TON       T1068 15	// R_1st DIE FPCB ALIGN BACKWARD
; L123
LOAD      P00062	// R_1st DIE ALIGN FORWARD
TON       T1069 20	// R_1st DIE ALIGN FORWARD
// ======================== VACUUM ALARM ==========================
; L125
LOAD      M12580	// R_1st MAND CYCLE RUN
AND       M12692	// R_1st MAND AUAc ¥ìe¨úi¢¯E
AND       P00140	// R_1st DIE VACUUM EJECTOR ON
AND NOT   M06611	// R_1st DIE VACUUM CHECK ON
AND       P0005D	// R_P&P UP (SENSOR)
AND       M01420	// R_PP 1 VC KP
AND NOT   M1902F	// DRY RUN
OUT       M12610	// R_1st DIE AUAc ¨úE©øN¨úi¢¯E
; L126
LOAD      M12580	// R_1st MAND CYCLE RUN
AND       P00140	// R_1st DIE VACUUM EJECTOR ON
AND NOT   M06611	// R_1st DIE VACUUM CHECK ON
AND       T1065	// R_P&P UP
AND NOT   M1902F	// DRY RUN
OUT       M12612	// R_1st DIE VC ALARM
; L127
LOAD      M12612	// R_1st DIE VC ALARM
OR        M12614	// R_1st DIE VC ALARM KP
AND       P00140	// R_1st DIE VACUUM EJECTOR ON
AND       P00013	// RIGHT DOOR OPEN
AND NOT   M06611	// R_1st DIE VACUUM CHECK ON
OUT       M12614	// R_1st DIE VC ALARM KP
; L129
LOADP     M00211	// RT_AUTO RUN
OR        M1261A	// R_1st DIE VC CLEAR OFF
AND       P00140	// R_1st DIE VACUUM EJECTOR ON
OUT       M1261A	// R_1st DIE VC CLEAR OFF

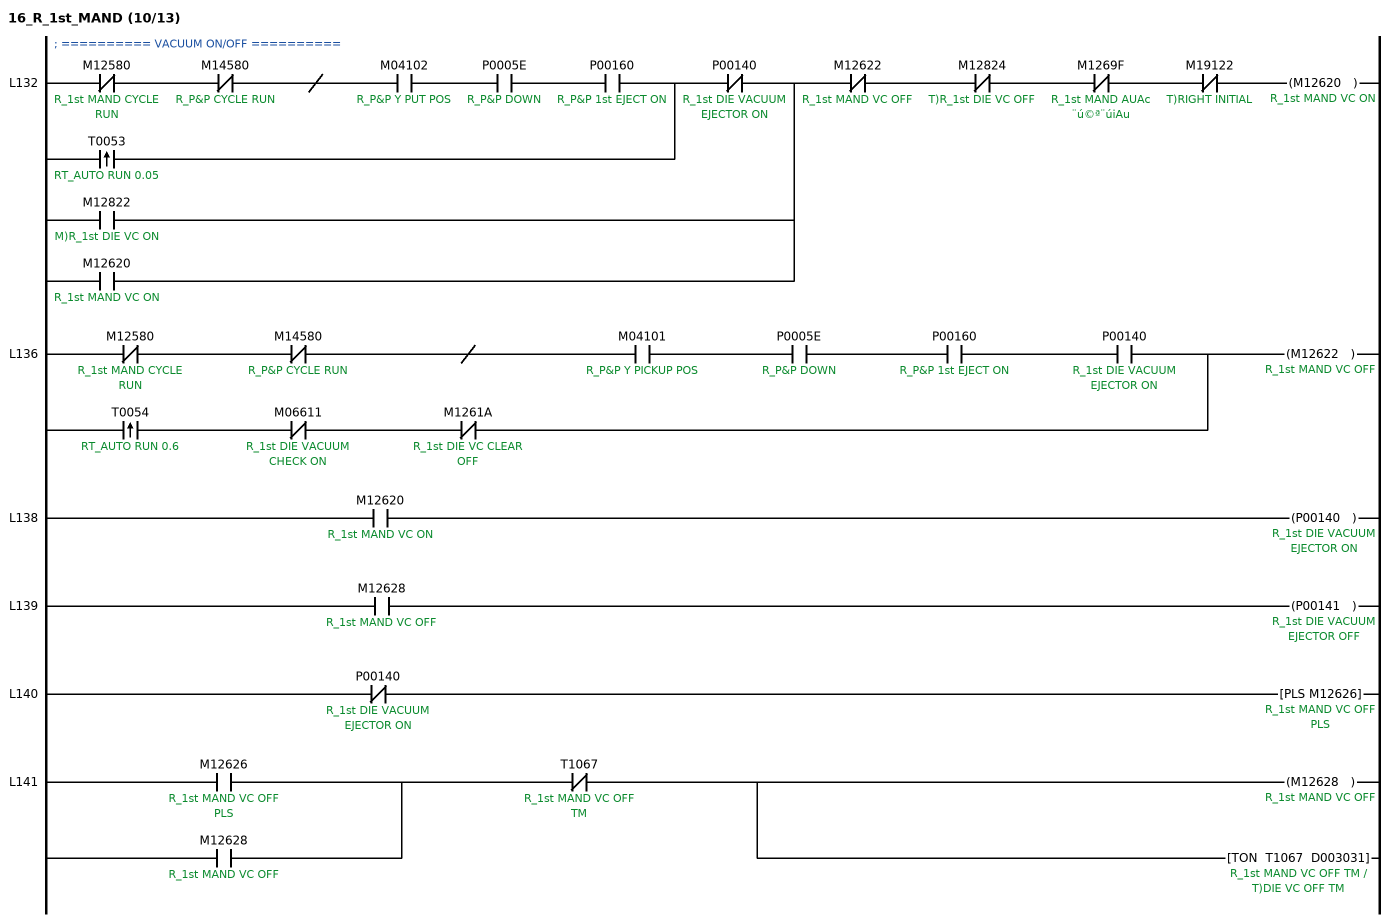
// ========== VACUUM ON/OFF ==========
; L132
LOAD NOT  M12580	// R_1st MAND CYCLE RUN
AND NOT   M14580	// R_P&P CYCLE RUN
NOT
AND       M04102	// R_P&P Y PUT POS
AND       P0005E	// R_P&P DOWN
AND       P00160	// R_P&P 1st EJECT ON
ORP       T0053	// RT_AUTO RUN 0.05
AND NOT   P00140	// R_1st DIE VACUUM EJECTOR ON
OR        M12822	// M)R_1st DIE VC ON
OR        M12620	// R_1st MAND VC ON
AND NOT   M12622	// R_1st MAND VC OFF
AND NOT   M12824	// T)R_1st DIE VC OFF
AND NOT   M1269F	// R_1st MAND AUAc ¨ú©ª¨úiAu
AND NOT   M19122	// T)RIGHT INITIAL
OUT       M12620	// R_1st MAND VC ON
; L136
LOAD NOT  M12580	// R_1st MAND CYCLE RUN
AND NOT   M14580	// R_P&P CYCLE RUN
NOT
AND       M04101	// R_P&P Y PICKUP POS
AND       P0005E	// R_P&P DOWN
AND       P00160	// R_P&P 1st EJECT ON
AND       P00140	// R_1st DIE VACUUM EJECTOR ON
LOADP     T0054	// RT_AUTO RUN 0.6
AND NOT   M06611	// R_1st DIE VACUUM CHECK ON
AND NOT   M1261A	// R_1st DIE VC CLEAR OFF
OR LOAD
OUT       M12622	// R_1st MAND VC OFF
; L138
LOAD      M12620	// R_1st MAND VC ON
OUT       P00140	// R_1st DIE VACUUM EJECTOR ON
; L139
LOAD      M12628	// R_1st MAND VC OFF
OUT       P00141	// R_1st DIE VACUUM EJECTOR OFF
; L140
LOAD NOT  P00140	// R_1st DIE VACUUM EJECTOR ON
OUTP      M12626	// R_1st MAND VC OFF PLS
; L141
LOAD      M12626	// R_1st MAND VC OFF PLS
OR        M12628	// R_1st MAND VC OFF
AND NOT   T1067	// R_1st MAND VC OFF TM
OUT       M12628	// R_1st MAND VC OFF
TON       T1067 D003031	// R_1st MAND VC OFF TM / T)DIE VC OFF TM

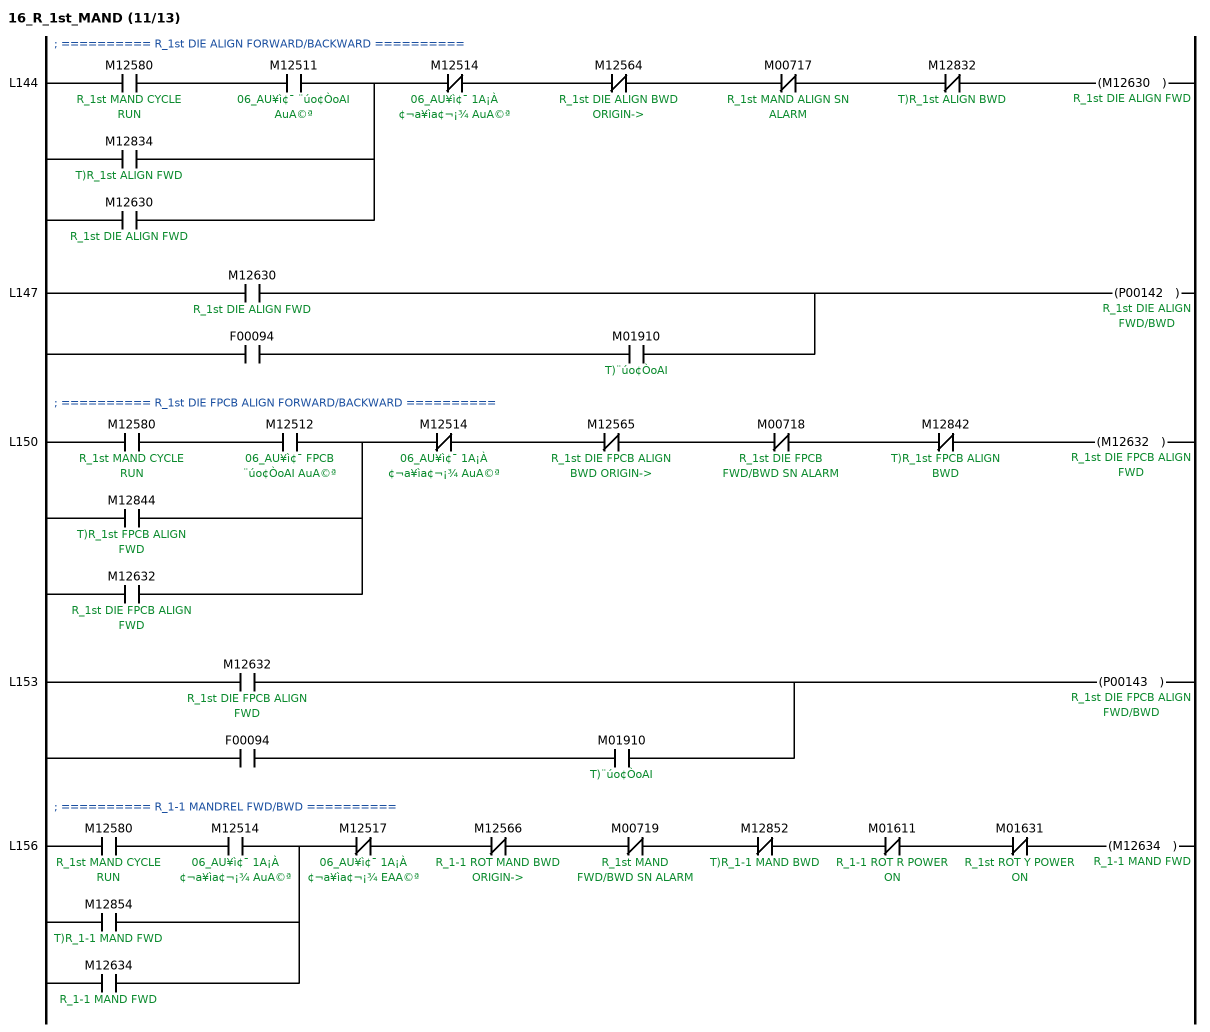
// ========== R_1st DIE ALIGN FORWARD/BACKWARD ==========
; L144
LOAD      M12580	// R_1st MAND CYCLE RUN
AND       M12511	// 06_AU¥ì¢¯ ¨úo¢ÒoAI AuA©ª
OR        M12834	// T)R_1st ALIGN FWD
OR        M12630	// R_1st DIE ALIGN FWD
AND NOT   M12514	// 06_AU¥ì¢¯ 1A¡À ¢¬a¥ìa¢¬¡¾ AuA©ª
AND NOT   M12564	// R_1st DIE ALIGN BWD ORIGIN->
AND NOT   M00717	// R_1st MAND ALIGN SN ALARM
AND NOT   M12832	// T)R_1st ALIGN BWD
OUT       M12630	// R_1st DIE ALIGN FWD
; L147
LOAD      M12630	// R_1st DIE ALIGN FWD
LOAD      F00094
AND       M01910	// T)¨úo¢ÒoAI
OR LOAD
OUT       P00142	// R_1st DIE ALIGN FWD/BWD
// ========== R_1st DIE FPCB ALIGN FORWARD/BACKWARD ==========
; L150
LOAD      M12580	// R_1st MAND CYCLE RUN
AND       M12512	// 06_AU¥ì¢¯ FPCB ¨úo¢ÒoAI AuA©ª
OR        M12844	// T)R_1st FPCB ALIGN FWD
OR        M12632	// R_1st DIE FPCB ALIGN FWD
AND NOT   M12514	// 06_AU¥ì¢¯ 1A¡À ¢¬a¥ìa¢¬¡¾ AuA©ª
AND NOT   M12565	// R_1st DIE FPCB ALIGN BWD ORIGIN->
AND NOT   M00718	// R_1st DIE FPCB FWD/BWD SN ALARM
AND NOT   M12842	// T)R_1st FPCB ALIGN BWD
OUT       M12632	// R_1st DIE FPCB ALIGN FWD
; L153
LOAD      M12632	// R_1st DIE FPCB ALIGN FWD
LOAD      F00094
AND       M01910	// T)¨úo¢ÒoAI
OR LOAD
OUT       P00143	// R_1st DIE FPCB ALIGN FWD/BWD
// ========== R_1-1 MANDREL FWD/BWD ==========
; L156
LOAD      M12580	// R_1st MAND CYCLE RUN
AND       M12514	// 06_AU¥ì¢¯ 1A¡À ¢¬a¥ìa¢¬¡¾ AuA©ª
OR        M12854	// T)R_1-1 MAND FWD
OR        M12634	// R_1-1 MAND FWD
AND NOT   M12517	// 06_AU¥ì¢¯ 1A¡À ¢¬a¥ìa¢¬¡¾ EAA©ª
AND NOT   M12566	// R_1-1 ROT MAND BWD ORIGIN->
AND NOT   M00719	// R_1st MAND FWD/BWD SN ALARM
AND NOT   M12852	// T)R_1-1 MAND BWD
AND NOT   M01611	// R_1-1 ROT R POWER ON
AND NOT   M01631	// R_1st ROT Y POWER ON
OUT       M12634	// R_1-1 MAND FWD

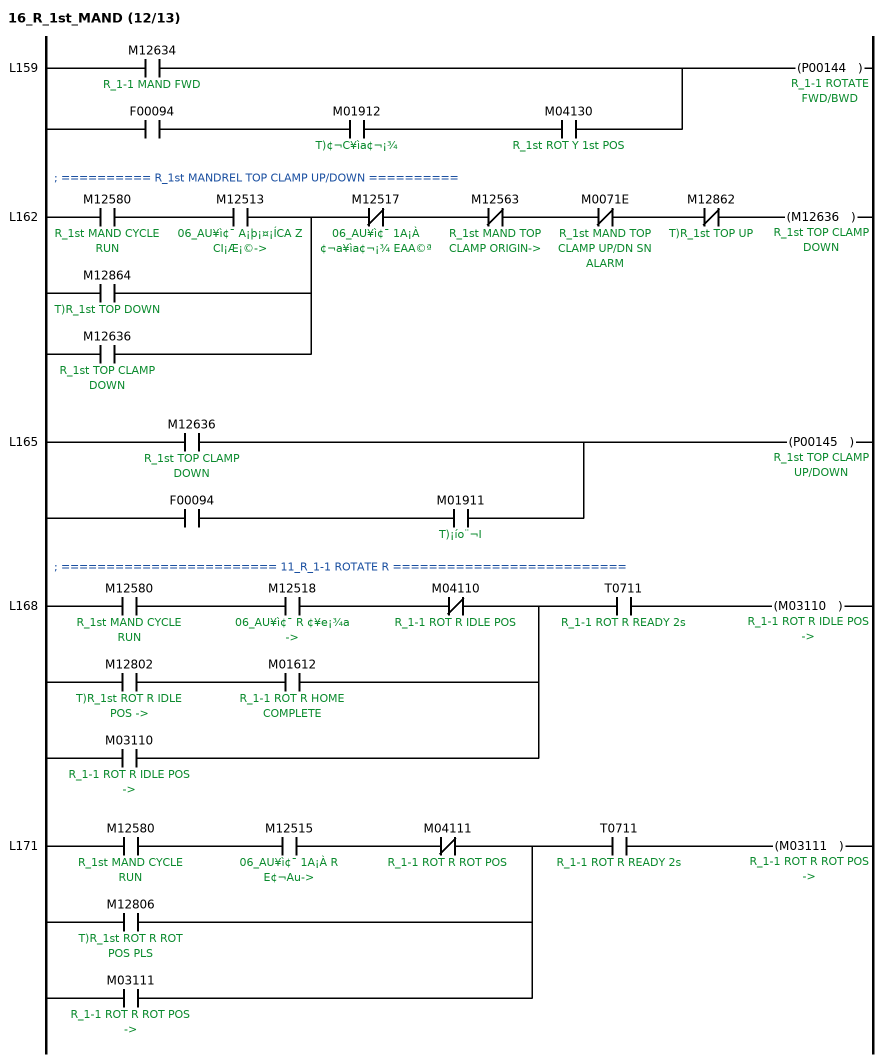
; L159
LOAD      M12634	// R_1-1 MAND FWD
LOAD      F00094
AND       M01912	// T)¢¬C¥ìa¢¬¡¾
AND       M04130	// R_1st ROT Y 1st POS
OR LOAD
OUT       P00144	// R_1-1 ROTATE FWD/BWD
// ========== R_1st MANDREL TOP CLAMP UP/DOWN ==========
; L162
LOAD      M12580	// R_1st MAND CYCLE RUN
AND       M12513	// 06_AU¥ì¢¯ A¡þ¡¤¡ÍCA Z CI¡Æ¡©->
OR        M12864	// T)R_1st TOP DOWN
OR        M12636	// R_1st TOP CLAMP DOWN
AND NOT   M12517	// 06_AU¥ì¢¯ 1A¡À ¢¬a¥ìa¢¬¡¾ EAA©ª
AND NOT   M12563	// R_1st MAND TOP CLAMP ORIGIN->
AND NOT   M0071E	// R_1st MAND TOP CLAMP UP/DN SN ALARM
AND NOT   M12862	// T)R_1st TOP UP
OUT       M12636	// R_1st TOP CLAMP DOWN
; L165
LOAD      M12636	// R_1st TOP CLAMP DOWN
LOAD      F00094
AND       M01911	// T)¡ío¨¬I
OR LOAD
OUT       P00145	// R_1st TOP CLAMP UP/DOWN
// ======================== 11_R_1-1 ROTATE R ==========================
; L168
LOAD      M12580	// R_1st MAND CYCLE RUN
AND       M12518	// 06_AU¥ì¢¯ R ¢¥e¡¾a ->
AND NOT   M04110	// R_1-1 ROT R IDLE POS
LOAD      M12802	// T)R_1st ROT R IDLE POS ->
AND       M01612	// R_1-1 ROT R HOME COMPLETE
OR LOAD
OR        M03110	// R_1-1 ROT R IDLE POS ->
AND       T0711	// R_1-1 ROT R READY 2s
OUT       M03110	// R_1-1 ROT R IDLE POS ->
; L171
LOAD      M12580	// R_1st MAND CYCLE RUN
AND       M12515	// 06_AU¥ì¢¯ 1A¡À R E¢¬Au->
AND NOT   M04111	// R_1-1 ROT R ROT POS
OR        M12806	// T)R_1st ROT R ROT POS PLS
OR        M03111	// R_1-1 ROT R ROT POS ->
AND       T0711	// R_1-1 ROT R READY 2s
OUT       M03111	// R_1-1 ROT R ROT POS ->

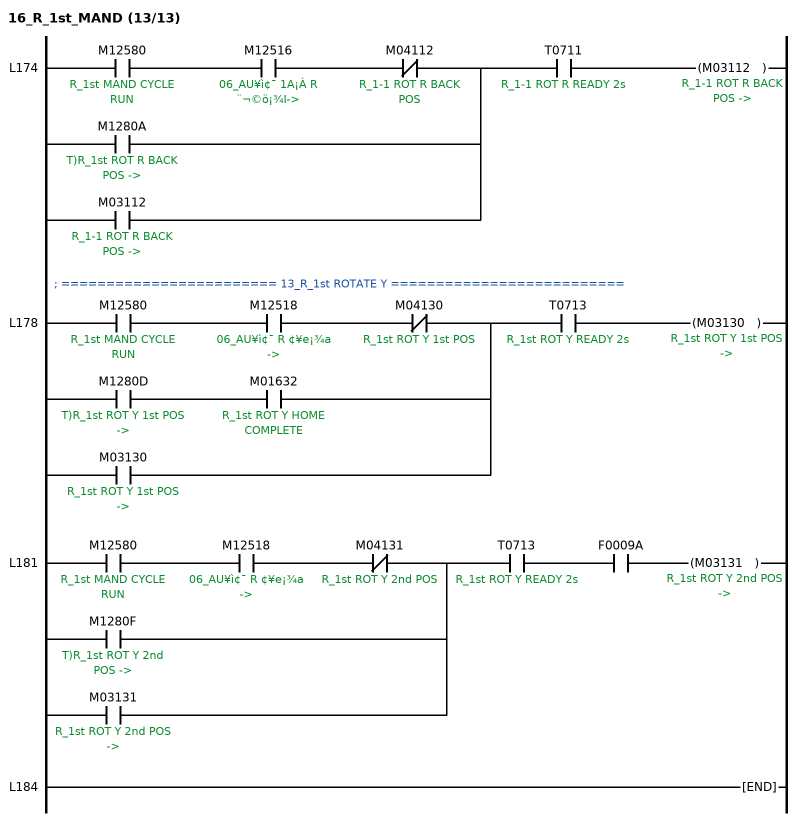
; L174
LOAD      M12580	// R_1st MAND CYCLE RUN
AND       M12516	// 06_AU¥ì¢¯ 1A¡À R ¨¬©ö¡¾I->
AND NOT   M04112	// R_1-1 ROT R BACK POS
OR        M1280A	// T)R_1st ROT R BACK POS ->
OR        M03112	// R_1-1 ROT R BACK POS ->
AND       T0711	// R_1-1 ROT R READY 2s
OUT       M03112	// R_1-1 ROT R BACK POS ->
// ======================== 13_R_1st ROTATE Y ==========================
; L178
LOAD      M12580	// R_1st MAND CYCLE RUN
AND       M12518	// 06_AU¥ì¢¯ R ¢¥e¡¾a ->
AND NOT   M04130	// R_1st ROT Y 1st POS
LOAD      M1280D	// T)R_1st ROT Y 1st POS ->
AND       M01632	// R_1st ROT Y HOME COMPLETE
OR LOAD
OR        M03130	// R_1st ROT Y 1st POS ->
AND       T0713	// R_1st ROT Y READY 2s
OUT       M03130	// R_1st ROT Y 1st POS ->
; L181
LOAD      M12580	// R_1st MAND CYCLE RUN
AND       M12518	// 06_AU¥ì¢¯ R ¢¥e¡¾a ->
AND NOT   M04131	// R_1st ROT Y 2nd POS
OR        M1280F	// T)R_1st ROT Y 2nd POS ->
OR        M03131	// R_1st ROT Y 2nd POS ->
AND       T0713	// R_1st ROT Y READY 2s
AND       F0009A
OUT       M03131	// R_1st ROT Y 2nd POS ->
; L184
END

PROGRAM 17_R_2nd_MAND (task: ¨ö¨¬A¥ì CA¡¤I¡¾¡¿¡¤¡Í)

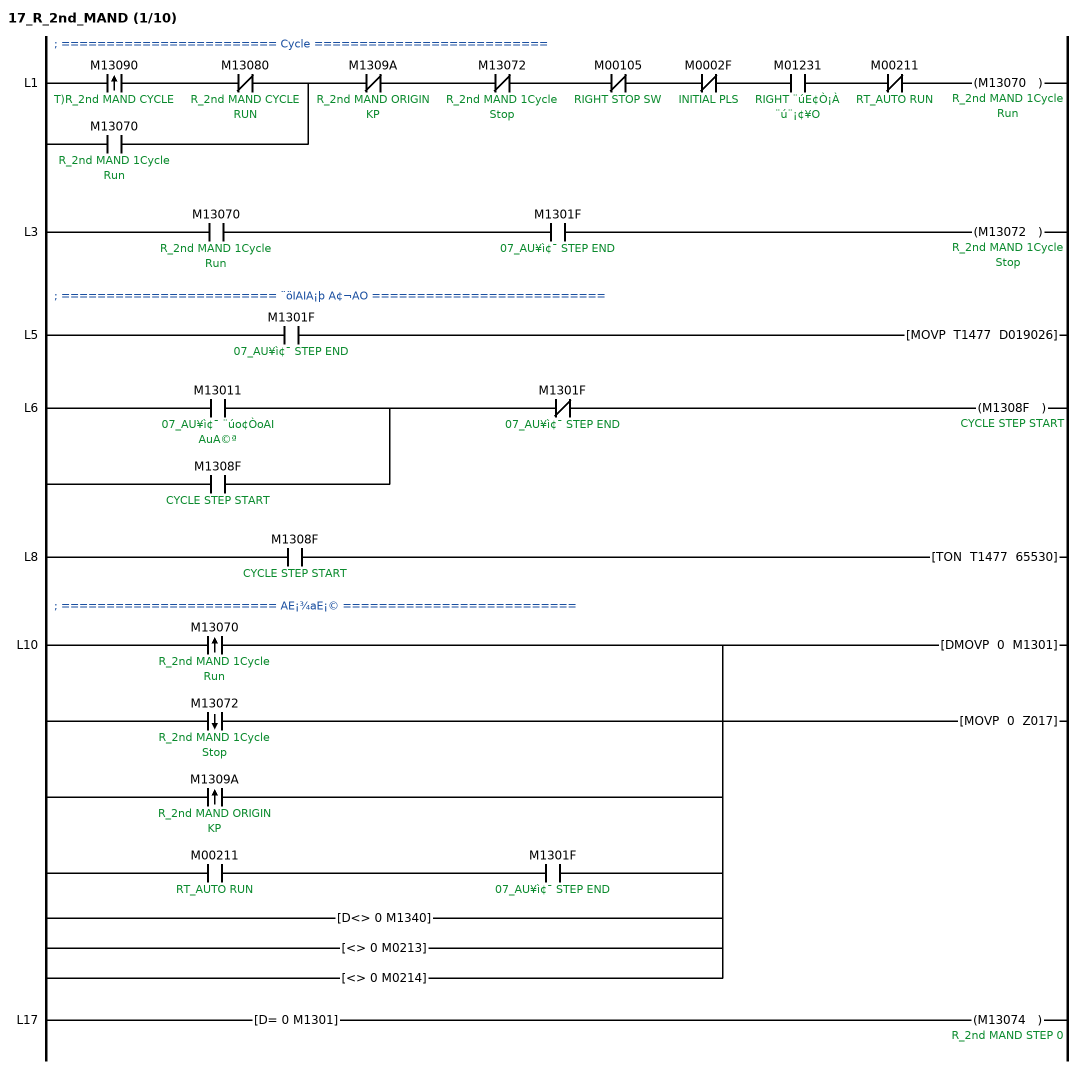
// ======================== Cycle ==========================
; L1
LOADP     M13090	// T)R_2nd MAND CYCLE
AND NOT   M13080	// R_2nd MAND CYCLE RUN
OR        M13070	// R_2nd MAND 1Cycle Run
AND NOT   M1309A	// R_2nd MAND ORIGIN KP
AND NOT   M13072	// R_2nd MAND 1Cycle Stop
AND NOT   M00105	// RIGHT STOP SW
AND NOT   M0002F	// INITIAL PLS
AND       M01231	// RIGHT ¨úE¢Ò¡À ¨ú¨¡¢¥O
AND NOT   M00211	// RT_AUTO RUN
OUT       M13070	// R_2nd MAND 1Cycle Run
; L3
LOAD      M13070	// R_2nd MAND 1Cycle Run
AND       M1301F	// 07_AU¥ì¢¯ STEP END
OUT       M13072	// R_2nd MAND 1Cycle Stop
// ======================== ¨öIAIA¡þ A¢¬AO ==========================
; L5
LOAD      M1301F	// 07_AU¥ì¢¯ STEP END
MOVP      T1477 D019026
; L6
LOAD      M13011	// 07_AU¥ì¢¯ ¨úo¢ÒoAI AuA©ª
OR        M1308F	// CYCLE STEP START
AND NOT   M1301F	// 07_AU¥ì¢¯ STEP END
OUT       M1308F	// CYCLE STEP START
; L8
LOAD      M1308F	// CYCLE STEP START
TON       T1477 65530
// ======================== AE¡¾aE¡© ==========================
; L10
LOADP     M13070	// R_2nd MAND 1Cycle Run
ORN       M13072	// R_2nd MAND 1Cycle Stop
ORP       M1309A	// R_2nd MAND ORIGIN KP
LOAD      M00211	// RT_AUTO RUN
AND       M1301F	// 07_AU¥ì¢¯ STEP END
OR LOAD
ORD<>     0 M1340
OR<>      0 M0213
OR<>      0 M0214
DMOVP     0 M1301
MOVP      0 Z017
; L17
LOADD=    0 M1301
OUT       M13074	// R_2nd MAND STEP 0

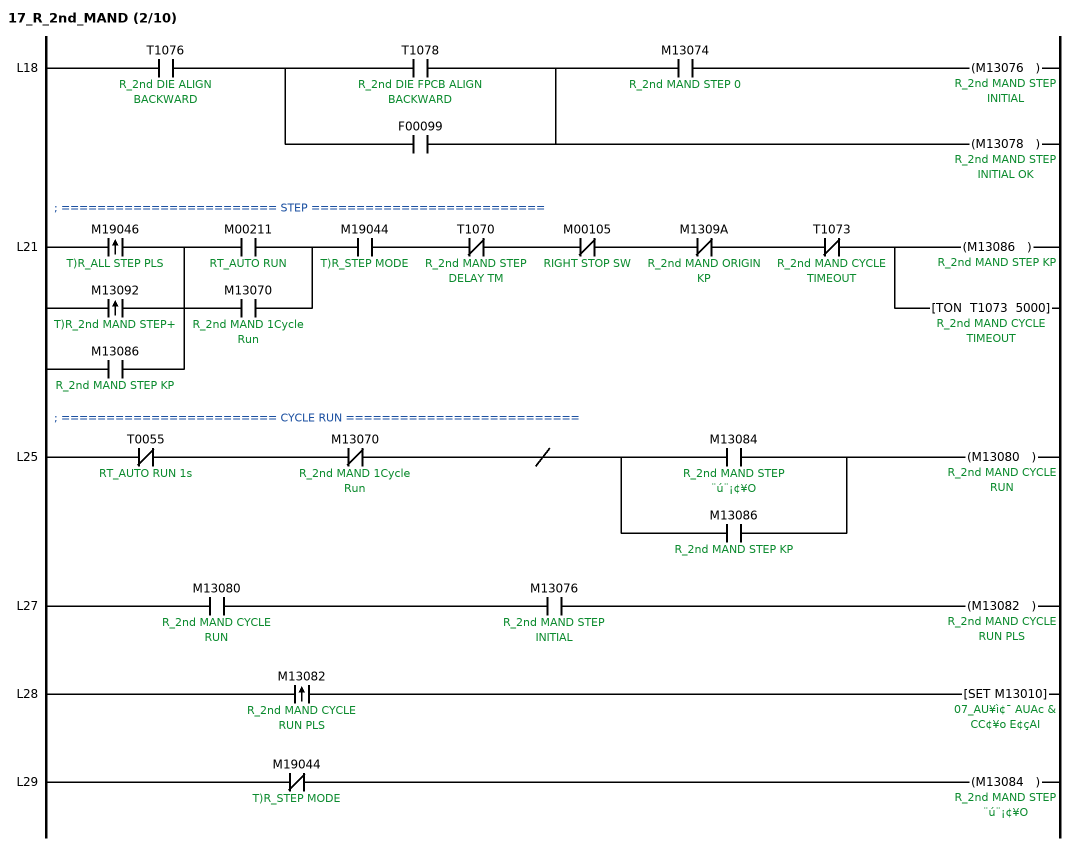
; L18
LOAD      T1076	// R_2nd DIE ALIGN BACKWARD
LOAD      T1078	// R_2nd DIE FPCB ALIGN BACKWARD
OR        F00099
AND LOAD
MPUSH
AND       M13074	// R_2nd MAND STEP 0
OUT       M13076	// R_2nd MAND STEP INITIAL
MPOP
OUT       M13078	// R_2nd MAND STEP INITIAL OK
// ======================== STEP ==========================
; L21
LOADP     M19046	// T)R_ALL STEP PLS
ORP       M13092	// T)R_2nd MAND STEP+
OR        M13086	// R_2nd MAND STEP KP
LOAD      M00211	// RT_AUTO RUN
OR        M13070	// R_2nd MAND 1Cycle Run
AND LOAD
AND       M19044	// T)R_STEP MODE
AND NOT   T1070	// R_2nd MAND STEP DELAY TM
AND NOT   M00105	// RIGHT STOP SW
AND NOT   M1309A	// R_2nd MAND ORIGIN KP
AND NOT   T1073	// R_2nd MAND CYCLE TIMEOUT
OUT       M13086	// R_2nd MAND STEP KP
TON       T1073 5000	// R_2nd MAND CYCLE TIMEOUT
// ======================== CYCLE RUN ==========================
; L25
LOAD NOT  T0055	// RT_AUTO RUN 1s
AND NOT   M13070	// R_2nd MAND 1Cycle Run
NOT
LOAD      M13084	// R_2nd MAND STEP ¨ú¨¡¢¥O
OR        M13086	// R_2nd MAND STEP KP
AND LOAD
OUT       M13080	// R_2nd MAND CYCLE RUN
; L27
LOAD      M13080	// R_2nd MAND CYCLE RUN
AND       M13076	// R_2nd MAND STEP INITIAL
OUT       M13082	// R_2nd MAND CYCLE RUN PLS
; L28
LOADP     M13082	// R_2nd MAND CYCLE RUN PLS
SET       M13010	// 07_AU¥ì¢¯ AUAc & CC¢¥o E¢çAI
; L29
LOAD NOT  M19044	// T)R_STEP MODE
OUT       M13084	// R_2nd MAND STEP ¨ú¨¡¢¥O

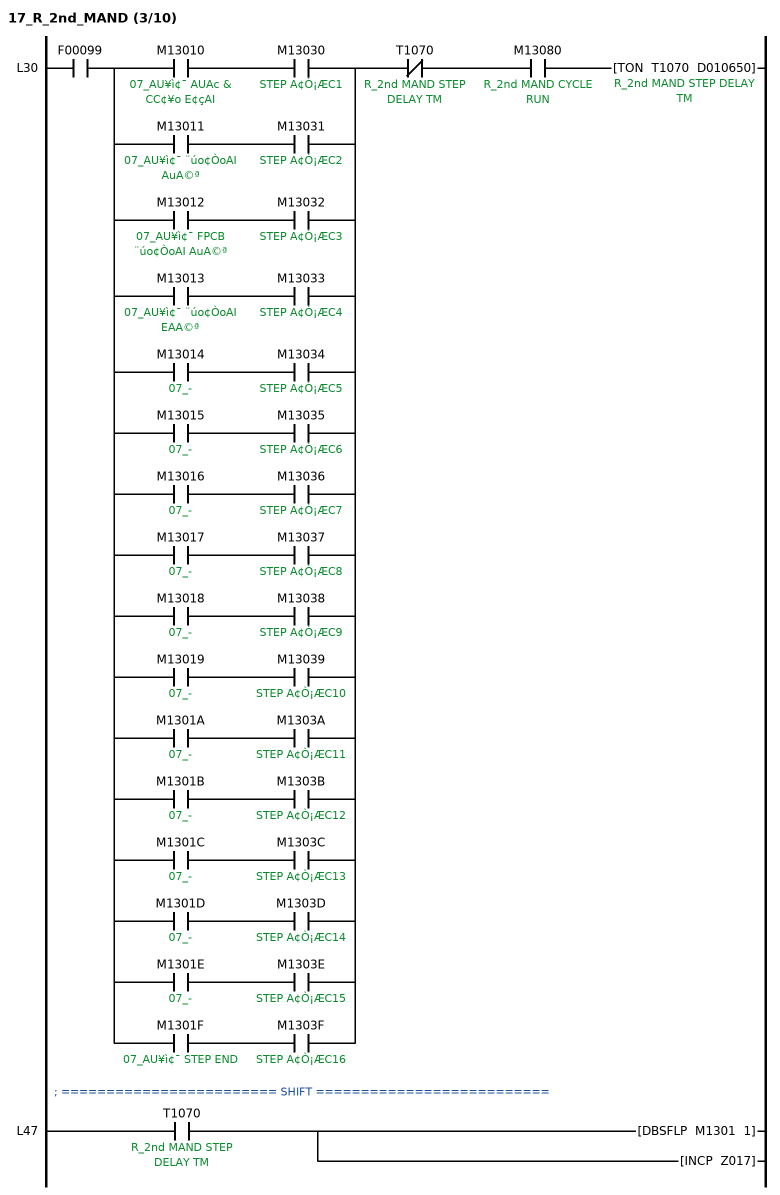
; L30
LOAD      F00099
LOAD      M13010	// 07_AU¥ì¢¯ AUAc & CC¢¥o E¢çAI
AND       M13030	// STEP A¢Ò¡ÆC1
LOAD      M13011	// 07_AU¥ì¢¯ ¨úo¢ÒoAI AuA©ª
AND       M13031	// STEP A¢Ò¡ÆC2
OR LOAD
LOAD      M13012	// 07_AU¥ì¢¯ FPCB ¨úo¢ÒoAI AuA©ª
AND       M13032	// STEP A¢Ò¡ÆC3
OR LOAD
LOAD      M13013	// 07_AU¥ì¢¯ ¨úo¢ÒoAI EAA©ª
AND       M13033	// STEP A¢Ò¡ÆC4
OR LOAD
LOAD      M13014	// 07_-
AND       M13034	// STEP A¢Ò¡ÆC5
OR LOAD
LOAD      M13015	// 07_-
AND       M13035	// STEP A¢Ò¡ÆC6
OR LOAD
LOAD      M13016	// 07_-
AND       M13036	// STEP A¢Ò¡ÆC7
OR LOAD
LOAD      M13017	// 07_-
AND       M13037	// STEP A¢Ò¡ÆC8
OR LOAD
LOAD      M13018	// 07_-
AND       M13038	// STEP A¢Ò¡ÆC9
OR LOAD
LOAD      M13019	// 07_-
AND       M13039	// STEP A¢Ò¡ÆC10
OR LOAD
LOAD      M1301A	// 07_-
AND       M1303A	// STEP A¢Ò¡ÆC11
OR LOAD
LOAD      M1301B	// 07_-
AND       M1303B	// STEP A¢Ò¡ÆC12
OR LOAD
LOAD      M1301C	// 07_-
AND       M1303C	// STEP A¢Ò¡ÆC13
OR LOAD
LOAD      M1301D	// 07_-
AND       M1303D	// STEP A¢Ò¡ÆC14
OR LOAD
LOAD      M1301E	// 07_-
AND       M1303E	// STEP A¢Ò¡ÆC15
OR LOAD
LOAD      M1301F	// 07_AU¥ì¢¯ STEP END
AND       M1303F	// STEP A¢Ò¡ÆC16
OR LOAD
AND LOAD
AND NOT   T1070	// R_2nd MAND STEP DELAY TM
AND       M13080	// R_2nd MAND CYCLE RUN
TON       T1070 D010650	// R_2nd MAND STEP DELAY TM
// ======================== SHIFT ==========================
; L47
LOAD      T1070	// R_2nd MAND STEP DELAY TM
DBSFLP    M1301 1
INCP      Z017

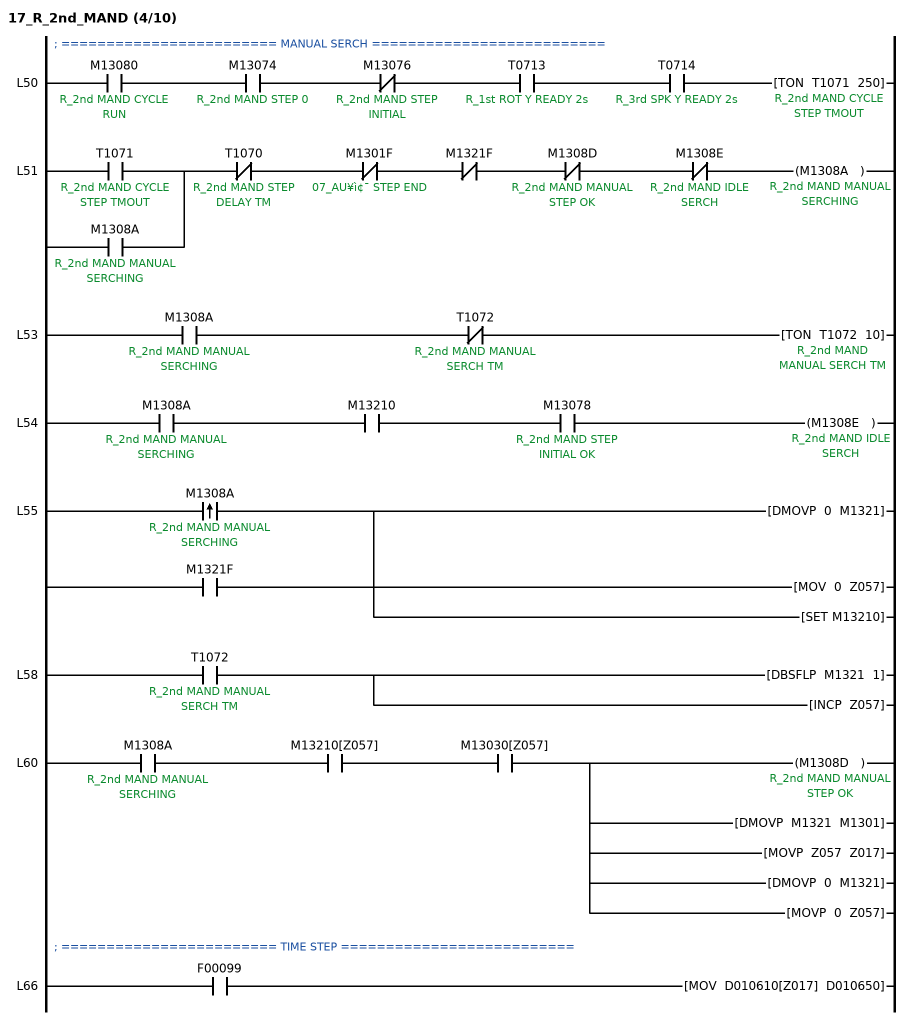
// ======================== MANUAL SERCH ==========================
; L50
LOAD      M13080	// R_2nd MAND CYCLE RUN
AND       M13074	// R_2nd MAND STEP 0
AND NOT   M13076	// R_2nd MAND STEP INITIAL
AND       T0713	// R_1st ROT Y READY 2s
AND       T0714	// R_3rd SPK Y READY 2s
TON       T1071 250	// R_2nd MAND CYCLE STEP TMOUT
; L51
LOAD      T1071	// R_2nd MAND CYCLE STEP TMOUT
OR        M1308A	// R_2nd MAND MANUAL SERCHING
AND NOT   T1070	// R_2nd MAND STEP DELAY TM
AND NOT   M1301F	// 07_AU¥ì¢¯ STEP END
AND NOT   M1321F
AND NOT   M1308D	// R_2nd MAND MANUAL STEP OK
AND NOT   M1308E	// R_2nd MAND IDLE SERCH
OUT       M1308A	// R_2nd MAND MANUAL SERCHING
; L53
LOAD      M1308A	// R_2nd MAND MANUAL SERCHING
AND NOT   T1072	// R_2nd MAND MANUAL SERCH TM
TON       T1072 10	// R_2nd MAND MANUAL SERCH TM
; L54
LOAD      M1308A	// R_2nd MAND MANUAL SERCHING
AND       M13210
AND       M13078	// R_2nd MAND STEP INITIAL OK
OUT       M1308E	// R_2nd MAND IDLE SERCH
; L55
LOADP     M1308A	// R_2nd MAND MANUAL SERCHING
OR        M1321F
DMOVP     0 M1321
MOV       0 Z057
SET       M13210
; L58
LOAD      T1072	// R_2nd MAND MANUAL SERCH TM
DBSFLP    M1321 1
INCP      Z057
; L60
LOAD      M1308A	// R_2nd MAND MANUAL SERCHING
AND       M13210[Z057]
AND       M13030[Z057]
OUT       M1308D	// R_2nd MAND MANUAL STEP OK
DMOVP     M1321 M1301
MOVP      Z057 Z017
DMOVP     0 M1321
MOVP      0 Z057
// ======================== TIME STEP ==========================
; L66
LOAD      F00099
MOV       D010610[Z017] D010650

